  MoveL 7660 to (-403.64, 335.28, -48.3) mm, rotated rx -180 ry 0 rz 0.01 deg; joints [35.458, -30.408, 74.668, -134.792, 54.854, 150.831]
  MoveL 7661 to (-403.75, 334.45, -48.33) mm, rotated rx -180 ry 0 rz 0.01 deg; joints [35.434, -30.43, 74.717, -134.831, 54.861, 150.87]
  MoveL 7662 to (-403.78, 333.95, -48.34) mm, rotated rx -180 ry 0 rz 0.01 deg; joints [35.42, -30.445, 74.752, -134.855, 54.867, 150.895]
  MoveL 7663 to (-403.79, 333.65, -48.35) mm, rotated rx -180 ry 0 rz 0.01 deg; joints [35.412, -30.454, 74.772, -134.869, 54.871, 150.909]
  MoveL 7664 to (-403.79, 333.1, -48.37) mm, rotated rx -180 ry 0 rz 0.01 deg; joints [35.398, -30.473, 74.813, -134.896, 54.879, 150.938]
  MoveL 7665 to (-401.27, 328.17, -48.57) mm, rotated rx -180 ry 0 rz 0.01 deg; joints [35.314, -30.758, 75.431, -135.148, 55.073, 151.276]
  MoveL 7666 to (-395.8, 327.3, -48.77) mm, rotated rx 180 ry 0 rz 0.01 deg; joints [35.394, -31.047, 76.052, -135.227, 55.349, 151.512]
  MoveL 7667 to (-391.89, 331.22, -48.97) mm, rotated rx 180 ry 0 rz 0.01 deg; joints [35.572, -31.096, 76.166, -135.071, 55.483, 151.459]
  MoveL 7668 to (-392.75, 336.69, -49.18) mm, rotated rx -180 ry 0 rz 0.01 deg; joints [35.7, -30.858, 75.678, -134.814, 55.371, 151.167]
  MoveL 7669 to (-397.69, 339.2, -49.38) mm, rotated rx 180 ry 0 rz 0.01 deg; joints [35.673, -30.52, 74.987, -134.669, 55.109, 150.878]
  MoveL 7670 to (-398.51, 339.2, -49.4) mm, rotated rx -180 ry 0 rz 0.01 deg; joints [35.658, -30.478, 74.902, -134.664, 55.071, 150.85]
  MoveL 7671 to (-399.34, 339.13, -49.43) mm, rotated rx 180 ry 0 rz 0.01 deg; joints [35.641, -30.438, 74.822, -134.661, 55.033, 150.826]
  MoveL 7672 to (-399.55, 339.1, -49.44) mm, rotated rx -180 ry 0 rz 0.01 deg; joints [35.636, -30.428, 74.802, -134.662, 55.024, 150.82]
  MoveL 7673 to (-402.87, 337.02, -49.58) mm, rotated rx -180 ry 0 rz 0.01 deg; joints [35.519, -30.33, 74.612, -134.739, 54.9, 150.812]
  MoveL 7674 to (-402.89, 336.99, -49.58) mm, rotated rx -180 ry 0 rz 0.01 deg; joints [35.517, -30.33, 74.612, -134.74, 54.899, 150.813]
  MoveL 7675 to (-403.36, 336.14, -49.62) mm, rotated rx 180 ry 0 rz 0.01 deg; joints [35.486, -30.334, 74.625, -134.777, 54.89, 150.84]
  MoveL 7676 to (-403.42, 336, -49.62) mm, rotated rx -180 ry 0 rz 0.01 deg; joints [35.482, -30.336, 74.629, -134.784, 54.889, 150.845]
  MoveL 7677 to (-403.6, 335.45, -49.64) mm, rotated rx -180 ry 0 rz 0.01 deg; joints [35.464, -30.345, 74.651, -134.809, 54.889, 150.867]
  MoveL 7678 to (-403.64, 335.28, -49.65) mm, rotated rx -180 ry 0 rz 0.01 deg; joints [35.459, -30.349, 74.659, -134.817, 54.889, 150.874]
  MoveL 7679 to (-403.75, 334.45, -49.68) mm, rotated rx -180 ry 0 rz 0.01 deg; joints [35.434, -30.371, 74.709, -134.856, 54.896, 150.913]
  MoveL 7680 to (-403.78, 333.95, -49.7) mm, rotated rx -180 ry 0 rz 0.01 deg; joints [35.421, -30.386, 74.743, -134.88, 54.903, 150.938]
  MoveL 7681 to (-403.79, 333.65, -49.71) mm, rotated rx 180 ry 0 rz 0.01 deg; joints [35.413, -30.396, 74.764, -134.894, 54.907, 150.952]
  MoveL 7682 to (-403.79, 333.1, -49.72) mm, rotated rx -180 ry 0 rz 0.01 deg; joints [35.398, -30.414, 74.804, -134.92, 54.915, 150.981]
  MoveL 7683 to (-401.27, 328.17, -49.93) mm, rotated rx 180 ry 0 rz 0.01 deg; joints [35.315, -30.699, 75.423, -135.172, 55.109, 151.319]
  MoveL 7684 to (-395.8, 327.3, -50.13) mm, rotated rx 180 ry 0 rz 0.01 deg; joints [35.395, -30.988, 76.044, -135.25, 55.385, 151.555]
  MoveL 7685 to (-391.89, 331.22, -50.33) mm, rotated rx 180 ry 0 rz 0.01 deg; joints [35.573, -31.037, 76.157, -135.095, 55.519, 151.502]
  MoveL 7686 to (-392.75, 336.69, -50.53) mm, rotated rx -180 ry 0 rz 0.01 deg; joints [35.701, -30.799, 75.67, -134.838, 55.407, 151.21]
  MoveL 7687 to (-397.69, 339.2, -50.73) mm, rotated rx 180 ry 0 rz 0.01 deg; joints [35.674, -30.461, 74.978, -134.693, 55.144, 150.921]
  MoveL 7688 to (-398.51, 339.2, -50.76) mm, rotated rx 180 ry 0 rz 0.01 deg; joints [35.659, -30.419, 74.894, -134.688, 55.106, 150.894]
  MoveL 7689 to (-399.34, 339.13, -50.79) mm, rotated rx -180 ry 0 rz 0.01 deg; joints [35.641, -30.379, 74.813, -134.686, 55.069, 150.869]
  MoveL 7690 to (-399.55, 339.1, -50.79) mm, rotated rx -180 ry 0 rz 0.01 deg; joints [35.636, -30.369, 74.793, -134.686, 55.059, 150.863]
  MoveL 7691 to (-402.87, 337.02, -50.93) mm, rotated rx -180 ry 0 rz 0.01 deg; joints [35.519, -30.271, 74.603, -134.763, 54.935, 150.855]
  MoveL 7692 to (-402.89, 336.99, -50.94) mm, rotated rx -180 ry 0 rz 0.01 deg; joints [35.518, -30.271, 74.603, -134.765, 54.935, 150.856]
  MoveL 7693 to (-403.36, 336.14, -50.97) mm, rotated rx 180 ry 0 rz 0.01 deg; joints [35.487, -30.276, 74.616, -134.802, 54.925, 150.883]
  MoveL 7694 to (-403.42, 336, -50.97) mm, rotated rx 180 ry 0 rz 0.01 deg; joints [35.482, -30.277, 74.62, -134.808, 54.924, 150.888]
  MoveL 7695 to (-403.6, 335.45, -50.99) mm, rotated rx -180 ry 0 rz 0.01 deg; joints [35.464, -30.287, 74.642, -134.833, 54.924, 150.91]
  MoveL 7696 to (-403.64, 335.28, -51) mm, rotated rx -180 ry 0 rz 0.01 deg; joints [35.459, -30.29, 74.651, -134.841, 54.925, 150.917]
  MoveL 7697 to (-403.75, 334.45, -51.03) mm, rotated rx -180 ry 0 rz 0.01 deg; joints [35.435, -30.312, 74.7, -134.88, 54.932, 150.956]
  MoveL 7698 to (-403.78, 333.95, -51.05) mm, rotated rx -180 ry 0 rz 0.01 deg; joints [35.421, -30.328, 74.734, -134.904, 54.938, 150.98]
  MoveL 7699 to (-403.79, 333.65, -51.06) mm, rotated rx 180 ry 0 rz 0.01 deg; joints [35.413, -30.337, 74.755, -134.918, 54.942, 150.995]
  MoveL 7700 to (-403.79, 333.1, -51.08) mm, rotated rx -180 ry 0 rz 0.01 deg; joints [35.399, -30.355, 74.795, -134.944, 54.951, 151.023]
  MoveL 7701 to (-401.27, 328.17, -51.28) mm, rotated rx 180 ry 0 rz 0.01 deg; joints [35.316, -30.64, 75.414, -135.197, 55.145, 151.362]
  MoveL 7702 to (-395.8, 327.3, -51.48) mm, rotated rx 180 ry 0 rz 0.01 deg; joints [35.396, -30.929, 76.035, -135.274, 55.421, 151.598]
  MoveL 7703 to (-391.89, 331.22, -51.68) mm, rotated rx -180 ry 0 rz 0.01 deg; joints [35.573, -30.978, 76.148, -135.118, 55.555, 151.545]
  MoveL 7704 to (-392.75, 336.69, -51.88) mm, rotated rx 180 ry 0 rz 0.01 deg; joints [35.702, -30.74, 75.661, -134.862, 55.443, 151.253]
  MoveL 7705 to (-397.69, 339.2, -52.08) mm, rotated rx -180 ry 0 rz 0.01 deg; joints [35.675, -30.402, 74.969, -134.717, 55.18, 150.964]
  MoveL 7706 to (-398.51, 339.2, -52.11) mm, rotated rx -180 ry 0 rz 0.01 deg; joints [35.659, -30.36, 74.885, -134.712, 55.142, 150.936]
  MoveL 7707 to (-399.34, 339.13, -52.14) mm, rotated rx -180 ry 0 rz 0.01 deg; joints [35.642, -30.32, 74.804, -134.71, 55.104, 150.912]
  MoveL 7708 to (-399.55, 339.1, -52.15) mm, rotated rx 180 ry 0 rz 0.01 deg; joints [35.637, -30.311, 74.784, -134.71, 55.095, 150.906]
  MoveL 7709 to (-402.87, 337.02, -52.29) mm, rotated rx 180 ry 0 rz 0.01 deg; joints [35.52, -30.212, 74.594, -134.788, 54.971, 150.898]
  MoveL 7710 to (-402.89, 336.99, -52.29) mm, rotated rx -180 ry 0 rz 0.01 deg; joints [35.519, -30.212, 74.594, -134.789, 54.97, 150.899]
  MoveL 7711 to (-403.36, 336.14, -52.32) mm, rotated rx 180 ry 0 rz 0.01 deg; joints [35.488, -30.217, 74.607, -134.826, 54.961, 150.926]
  MoveL 7712 to (-403.42, 336, -52.33) mm, rotated rx -180 ry 0 rz 0.01 deg; joints [35.483, -30.219, 74.611, -134.832, 54.96, 150.931]
  MoveL 7713 to (-403.6, 335.45, -52.35) mm, rotated rx 180 ry 0 rz 0.01 deg; joints [35.465, -30.228, 74.633, -134.857, 54.96, 150.953]
  MoveL 7714 to (-403.64, 335.28, -52.35) mm, rotated rx -180 ry 0 rz 0.01 deg; joints [35.46, -30.231, 74.642, -134.865, 54.96, 150.96]
  MoveL 7715 to (-403.75, 334.45, -52.38) mm, rotated rx -180 ry 0 rz 0.01 deg; joints [35.436, -30.253, 74.691, -134.904, 54.967, 150.999]
  MoveL 7716 to (-403.78, 333.95, -52.4) mm, rotated rx -180 ry 0 rz 0.01 deg; joints [35.422, -30.269, 74.725, -134.928, 54.974, 151.023]
  MoveL 7717 to (-403.79, 333.65, -52.41) mm, rotated rx -180 ry 0 rz 0.01 deg; joints [35.414, -30.278, 74.746, -134.942, 54.978, 151.038]
  MoveL 7718 to (-403.79, 333.1, -52.43) mm, rotated rx -180 ry 0 rz 0.01 deg; joints [35.399, -30.296, 74.786, -134.968, 54.986, 151.066]
  MoveL 7719 to (-401.27, 328.17, -52.63) mm, rotated rx 180 ry 0 rz 0.01 deg; joints [35.316, -30.581, 75.405, -135.22, 55.181, 151.405]
  MoveL 7720 to (-395.8, 327.3, -52.83) mm, rotated rx 180 ry 0 rz 0.01 deg; joints [35.396, -30.87, 76.026, -135.298, 55.457, 151.64]
  MoveL 7721 to (-391.89, 331.22, -53.03) mm, rotated rx -180 ry 0 rz 0.01 deg; joints [35.574, -30.918, 76.139, -135.142, 55.591, 151.588]
  MoveL 7722 to (-392.75, 336.69, -53.23) mm, rotated rx -180 ry 0 rz 0.01 deg; joints [35.702, -30.681, 75.652, -134.886, 55.478, 151.296]
  MoveL 7723 to (-397.69, 339.2, -53.43) mm, rotated rx -180 ry 0 rz 0.01 deg; joints [35.675, -30.343, 74.96, -134.741, 55.215, 151.007]
  MoveL 7724 to (-398.51, 339.2, -53.46) mm, rotated rx -180 ry 0 rz 0.01 deg; joints [35.66, -30.301, 74.876, -134.736, 55.177, 150.979]
  MoveL 7725 to (-399.34, 339.13, -53.49) mm, rotated rx 180 ry 0 rz 0.01 deg; joints [35.642, -30.261, 74.795, -134.734, 55.14, 150.954]
  MoveL 7726 to (-399.55, 339.1, -53.5) mm, rotated rx -180 ry 0 rz 0.01 deg; joints [35.637, -30.252, 74.775, -134.734, 55.13, 150.949]
  MoveL 7727 to (-402.87, 337.02, -53.64) mm, rotated rx -180 ry 0 rz 0.01 deg; joints [35.52, -30.154, 74.585, -134.812, 55.006, 150.941]
  MoveL 7728 to (-402.89, 336.99, -53.64) mm, rotated rx -180 ry 0 rz 0.01 deg; joints [35.519, -30.154, 74.585, -134.813, 55.005, 150.942]
  MoveL 7729 to (-403.36, 336.14, -53.67) mm, rotated rx -180 ry 0 rz 0.01 deg; joints [35.488, -30.158, 74.598, -134.85, 54.996, 150.968]
  MoveL 7730 to (-403.42, 336, -53.68) mm, rotated rx -180 ry 0 rz 0.01 deg; joints [35.483, -30.16, 74.602, -134.856, 54.995, 150.974]
  MoveL 7731 to (-403.6, 335.45, -53.7) mm, rotated rx 180 ry 0 rz 0.01 deg; joints [35.465, -30.169, 74.624, -134.881, 54.995, 150.995]
  MoveL 7732 to (-403.64, 335.28, -53.71) mm, rotated rx -180 ry 0 rz 0.01 deg; joints [35.46, -30.173, 74.633, -134.889, 54.996, 151.003]
  MoveL 7733 to (-403.75, 334.45, -53.74) mm, rotated rx -180 ry 0 rz 0.01 deg; joints [35.436, -30.194, 74.682, -134.928, 55.003, 151.041]
  MoveL 7734 to (-403.78, 333.95, -53.75) mm, rotated rx -180 ry 0 rz 0.01 deg; joints [35.422, -30.21, 74.716, -134.952, 55.009, 151.066]
  MoveL 7735 to (-403.79, 333.65, -53.76) mm, rotated rx -180 ry 0 rz 0.01 deg; joints [35.415, -30.219, 74.737, -134.966, 55.013, 151.081]
  MoveL 7736 to (-403.79, 333.1, -53.78) mm, rotated rx -180 ry 0 rz 0.01 deg; joints [35.4, -30.237, 74.777, -134.992, 55.022, 151.109]
  MoveL 7737 to (-401.27, 328.17, -53.98) mm, rotated rx -180 ry 0 rz 0.01 deg; joints [35.317, -30.522, 75.396, -135.244, 55.217, 151.447]
  MoveL 7738 to (-395.8, 327.3, -54.18) mm, rotated rx 180 ry 0 rz 0.01 deg; joints [35.397, -30.811, 76.017, -135.322, 55.493, 151.683]
  MoveL 7739 to (-391.89, 331.22, -54.38) mm, rotated rx 180 ry 0 rz 0.01 deg; joints [35.575, -30.859, 76.13, -135.166, 55.627, 151.63]
  MoveL 7740 to (-392.75, 336.69, -54.59) mm, rotated rx -180 ry 0 rz 0.01 deg; joints [35.703, -30.621, 75.643, -134.91, 55.514, 151.339]
  MoveL 7741 to (-397.69, 339.2, -54.79) mm, rotated rx -180 ry 0 rz 0.01 deg; joints [35.676, -30.284, 74.951, -134.765, 55.251, 151.05]
  MoveL 7742 to (-398.51, 339.2, -54.81) mm, rotated rx -180 ry 0 rz 0.01 deg; joints [35.66, -30.242, 74.866, -134.76, 55.213, 151.022]
  MoveL 7743 to (-399.34, 339.13, -54.84) mm, rotated rx -180 ry 0 rz 0.01 deg; joints [35.643, -30.202, 74.786, -134.758, 55.175, 150.997]
  MoveL 7744 to (-399.55, 339.1, -54.85) mm, rotated rx -180 ry 0 rz 0.01 deg; joints [35.638, -30.193, 74.766, -134.758, 55.165, 150.992]
  MoveL 7745 to (-402.87, 337.02, -54.99) mm, rotated rx 180 ry 0 rz 0.01 deg; joints [35.521, -30.095, 74.576, -134.836, 55.041, 150.984]
  MoveL 7746 to (-402.89, 336.99, -54.99) mm, rotated rx -180 ry 0 rz 0.01 deg; joints [35.52, -30.095, 74.576, -134.837, 55.041, 150.984]
  MoveL 7747 to (-403.36, 336.14, -55.03) mm, rotated rx -180 ry 0 rz 0.01 deg; joints [35.489, -30.099, 74.589, -134.874, 55.031, 151.011]
  MoveL 7748 to (-403.42, 336, -55.03) mm, rotated rx 180 ry 0 rz 0.01 deg; joints [35.484, -30.101, 74.593, -134.88, 55.031, 151.016]
  MoveL 7749 to (-403.6, 335.45, -55.05) mm, rotated rx 180 ry 0 rz 0.01 deg; joints [35.466, -30.11, 74.615, -134.905, 55.03, 151.038]
  MoveL 7750 to (-403.64, 335.28, -55.06) mm, rotated rx 180 ry 0 rz 0.01 deg; joints [35.461, -30.114, 74.623, -134.913, 55.031, 151.045]
  MoveL 7751 to (-403.75, 334.45, -55.09) mm, rotated rx -180 ry 0 rz 0.01 deg; joints [35.437, -30.135, 74.673, -134.952, 55.038, 151.084]
  MoveL 7752 to (-403.78, 333.95, -55.11) mm, rotated rx -180 ry 0 rz 0.01 deg; joints [35.423, -30.151, 74.707, -134.976, 55.045, 151.109]
  MoveL 7753 to (-403.79, 333.65, -55.12) mm, rotated rx -180 ry 0 rz 0.01 deg; joints [35.415, -30.16, 74.727, -134.99, 55.049, 151.123]
  MoveL 7754 to (-403.79, 333.1, -55.14) mm, rotated rx -180 ry 0 rz 0.01 deg; joints [35.401, -30.178, 74.768, -135.016, 55.057, 151.151]
  MoveL 7755 to (-401.27, 328.17, -55.34) mm, rotated rx -180 ry 0 rz 0.01 deg; joints [35.317, -30.463, 75.387, -135.268, 55.252, 151.49]
  MoveL 7756 to (-395.8, 327.3, -55.54) mm, rotated rx -180 ry 0 rz 0.01 deg; joints [35.397, -30.751, 76.008, -135.345, 55.529, 151.725]
  MoveL 7757 to (-391.89, 331.22, -55.74) mm, rotated rx -180 ry 0 rz 0.01 deg; joints [35.575, -30.8, 76.121, -135.189, 55.663, 151.673]
  MoveL 7758 to (-392.75, 336.69, -55.94) mm, rotated rx 180 ry 0 rz 0.01 deg; joints [35.703, -30.562, 75.633, -134.934, 55.55, 151.381]
  MoveL 7759 to (-397.69, 339.2, -56.14) mm, rotated rx -180 ry 0 rz 0.01 deg; joints [35.676, -30.225, 74.942, -134.789, 55.286, 151.092]
  MoveL 7760 to (-398.51, 339.2, -56.17) mm, rotated rx -180 ry 0 rz 0.01 deg; joints [35.661, -30.183, 74.857, -134.784, 55.248, 151.065]
  MoveL 7761 to (-399.34, 339.13, -56.2) mm, rotated rx 180 ry 0 rz 0.01 deg; joints [35.644, -30.143, 74.776, -134.782, 55.21, 151.04]
  MoveL 7762 to (-399.55, 339.1, -56.2) mm, rotated rx 180 ry 0 rz 0.01 deg; joints [35.639, -30.134, 74.756, -134.782, 55.201, 151.034]
  MoveL 7763 to (-402.87, 337.02, -56.34) mm, rotated rx -180 ry 0 rz 0.01 deg; joints [35.522, -30.036, 74.566, -134.86, 55.076, 151.026]
  MoveL 7764 to (-402.89, 336.99, -56.35) mm, rotated rx -180 ry 0 rz 0.01 deg; joints [35.52, -30.036, 74.566, -134.861, 55.076, 151.027]
  MoveL 7765 to (-403.36, 336.14, -56.38) mm, rotated rx -180 ry 0 rz 0.01 deg; joints [35.489, -30.04, 74.58, -134.898, 55.067, 151.054]
  MoveL 7766 to (-403.42, 336, -56.38) mm, rotated rx 180 ry 0 rz 0.01 deg; joints [35.484, -30.042, 74.584, -134.904, 55.066, 151.059]
  MoveL 7767 to (-403.6, 335.45, -56.4) mm, rotated rx -180 ry 0 rz 0.01 deg; joints [35.467, -30.051, 74.605, -134.929, 55.066, 151.08]
  MoveL 7768 to (-403.64, 335.28, -56.41) mm, rotated rx -180 ry 0 rz 0.01 deg; joints [35.461, -30.055, 74.614, -134.937, 55.066, 151.088]
  MoveL 7769 to (-403.75, 334.45, -56.44) mm, rotated rx -180 ry 0 rz 0.01 deg; joints [35.437, -30.076, 74.663, -134.976, 55.074, 151.126]
  MoveL 7770 to (-403.78, 333.95, -56.46) mm, rotated rx -180 ry 0 rz 0.01 deg; joints [35.424, -30.092, 74.697, -135, 55.08, 151.151]
  MoveL 7771 to (-403.79, 333.65, -56.47) mm, rotated rx -180 ry 0 rz 0.01 deg; joints [35.416, -30.101, 74.718, -135.014, 55.084, 151.166]
  MoveL 7772 to (-403.79, 333.1, -56.49) mm, rotated rx 180 ry 0 rz 0.01 deg; joints [35.401, -30.119, 74.758, -135.04, 55.093, 151.194]
  MoveL 7773 to (-401.27, 328.17, -56.69) mm, rotated rx 180 ry 0 rz 0.01 deg; joints [35.318, -30.404, 75.377, -135.292, 55.288, 151.532]
  MoveL 7774 to (-395.8, 327.3, -56.89) mm, rotated rx -180 ry 0 rz 0.01 deg; joints [35.398, -30.692, 75.998, -135.369, 55.565, 151.768]
  MoveL 7775 to (-391.89, 331.22, -57.09) mm, rotated rx 180 ry 0 rz 0.01 deg; joints [35.576, -30.74, 76.112, -135.213, 55.699, 151.715]
  MoveL 7776 to (-392.75, 336.69, -57.29) mm, rotated rx 180 ry 0 rz 0.01 deg; joints [35.704, -30.503, 75.624, -134.957, 55.585, 151.424]
  MoveL 7777 to (-397.69, 339.2, -57.49) mm, rotated rx -180 ry 0 rz 0.01 deg; joints [35.677, -30.166, 74.932, -134.813, 55.321, 151.135]
  MoveL 7778 to (-398.51, 339.2, -57.52) mm, rotated rx -180 ry 0 rz 0.01 deg; joints [35.661, -30.124, 74.847, -134.808, 55.283, 151.107]
  MoveL 7779 to (-399.34, 339.13, -57.55) mm, rotated rx 180 ry 0 rz 0.01 deg; joints [35.644, -30.084, 74.767, -134.806, 55.245, 151.082]
  MoveL 7780 to (-399.55, 339.1, -57.56) mm, rotated rx -180 ry 0 rz 0.01 deg; joints [35.639, -30.074, 74.747, -134.806, 55.236, 151.077]
  MoveL 7781 to (-402.87, 337.02, -57.7) mm, rotated rx -180 ry 0 rz 0.01 deg; joints [35.522, -29.976, 74.556, -134.884, 55.112, 151.068]
  MoveL 7782 to (-402.89, 336.99, -57.7) mm, rotated rx -180 ry 0 rz 0.01 deg; joints [35.521, -29.976, 74.556, -134.885, 55.111, 151.069]
  MoveL 7783 to (-403.36, 336.14, -57.73) mm, rotated rx -180 ry 0 rz 0.01 deg; joints [35.49, -29.981, 74.57, -134.922, 55.102, 151.096]
  MoveL 7784 to (-403.42, 336, -57.74) mm, rotated rx -180 ry 0 rz 0.01 deg; joints [35.485, -29.983, 74.574, -134.928, 55.101, 151.101]
  MoveL 7785 to (-403.6, 335.45, -57.76) mm, rotated rx -180 ry 0 rz 0.01 deg; joints [35.467, -29.992, 74.596, -134.953, 55.101, 151.123]
  MoveL 7786 to (-403.64, 335.28, -57.76) mm, rotated rx 180 ry 0 rz 0.01 deg; joints [35.462, -29.995, 74.604, -134.961, 55.102, 151.13]
  MoveL 7787 to (-403.75, 334.45, -57.79) mm, rotated rx -180 ry 0 rz 0.01 deg; joints [35.438, -30.017, 74.654, -135, 55.109, 151.169]
  MoveL 7788 to (-403.78, 333.95, -57.81) mm, rotated rx -180 ry 0 rz 0.01 deg; joints [35.424, -30.033, 74.688, -135.024, 55.115, 151.193]
  MoveL 7789 to (-403.79, 333.65, -57.82) mm, rotated rx -180 ry 0 rz 0.01 deg; joints [35.416, -30.042, 74.708, -135.038, 55.119, 151.208]
  MoveL 7790 to (-403.79, 333.1, -57.84) mm, rotated rx -180 ry 0 rz 0.01 deg; joints [35.402, -30.06, 74.749, -135.064, 55.128, 151.236]
  MoveL 7791 to (-401.27, 328.17, -58.04) mm, rotated rx -180 ry 0 rz 0.01 deg; joints [35.319, -30.344, 75.368, -135.315, 55.324, 151.574]
  MoveL 7792 to (-395.8, 327.3, -58.24) mm, rotated rx 180 ry 0 rz 0.01 deg; joints [35.399, -30.632, 75.989, -135.392, 55.601, 151.81]
  MoveL 7793 to (-391.89, 331.22, -58.44) mm, rotated rx -180 ry 0 rz 0.01 deg; joints [35.576, -30.681, 76.102, -135.236, 55.734, 151.757]
  MoveL 7794 to (-392.75, 336.69, -58.64) mm, rotated rx 180 ry 0 rz 0.01 deg; joints [35.705, -30.443, 75.614, -134.981, 55.621, 151.466]
  MoveL 7795 to (-397.69, 339.2, -58.84) mm, rotated rx 180 ry 0 rz 0.01 deg; joints [35.677, -30.106, 74.922, -134.836, 55.356, 151.177]
  MoveL 7796 to (-398.51, 339.2, -58.87) mm, rotated rx -180 ry 0 rz 0.01 deg; joints [35.662, -30.065, 74.838, -134.831, 55.318, 151.149]
  MoveL 7797 to (-399.34, 339.13, -58.9) mm, rotated rx -180 ry 0 rz 0.01 deg; joints [35.645, -30.025, 74.757, -134.829, 55.281, 151.125]
  MoveL 7798 to (-399.55, 339.1, -58.91) mm, rotated rx -180 ry 0 rz 0.01 deg; joints [35.64, -30.015, 74.737, -134.83, 55.271, 151.119]
  MoveL 7799 to (-402.87, 337.02, -59.05) mm, rotated rx 180 ry 0 rz 0.01 deg; joints [35.523, -29.917, 74.547, -134.907, 55.147, 151.111]
  MoveL 7800 to (-402.89, 336.99, -59.05) mm, rotated rx -180 ry 0 rz 0.01 deg; joints [35.522, -29.917, 74.547, -134.909, 55.146, 151.112]
  MoveL 7801 to (-403.36, 336.14, -59.08) mm, rotated rx -180 ry 0 rz 0.01 deg; joints [35.491, -29.922, 74.56, -134.946, 55.137, 151.138]
  MoveL 7802 to (-403.42, 336, -59.09) mm, rotated rx -180 ry 0 rz 0.01 deg; joints [35.486, -29.923, 74.564, -134.952, 55.136, 151.143]
  MoveL 7803 to (-403.6, 335.45, -59.11) mm, rotated rx -180 ry 0 rz 0.01 deg; joints [35.468, -29.933, 74.586, -134.977, 55.136, 151.165]
  MoveL 7804 to (-403.64, 335.28, -59.12) mm, rotated rx -180 ry 0 rz 0.01 deg; joints [35.463, -29.936, 74.594, -134.985, 55.137, 151.172]
  MoveL 7805 to (-403.75, 334.45, -59.15) mm, rotated rx -180 ry 0 rz 0.01 deg; joints [35.438, -29.958, 74.644, -135.024, 55.144, 151.211]
  MoveL 7806 to (-403.78, 333.95, -59.16) mm, rotated rx -180 ry 0 rz 0.01 deg; joints [35.425, -29.973, 74.678, -135.047, 55.151, 151.236]
  MoveL 7807 to (-403.79, 333.65, -59.17) mm, rotated rx -180 ry 0 rz 0.01 deg; joints [35.417, -29.983, 74.699, -135.061, 55.155, 151.25]
  MoveL 7808 to (-403.79, 333.1, -59.19) mm, rotated rx -180 ry 0 rz 0.01 deg; joints [35.402, -30.001, 74.739, -135.088, 55.163, 151.278]
  MoveL 7809 to (-401.27, 328.17, -59.39) mm, rotated rx 180 ry 0 rz 0.01 deg; joints [35.319, -30.285, 75.358, -135.339, 55.359, 151.616]
  MoveL 7810 to (-395.8, 327.3, -59.59) mm, rotated rx 180 ry 0 rz 0.01 deg; joints [35.399, -30.573, 75.979, -135.416, 55.636, 151.852]
  MoveL 7811 to (-391.89, 331.22, -59.79) mm, rotated rx 180 ry 0 rz 0.01 deg; joints [35.577, -30.621, 76.092, -135.259, 55.77, 151.8]
  MoveL 7812 to (-392.75, 336.69, -60) mm, rotated rx -180 ry 0 rz 0.01 deg; joints [35.705, -30.384, 75.604, -135.004, 55.656, 151.508]
  MoveL 7813 to (-397.69, 339.2, -60.2) mm, rotated rx -180 ry 0 rz 0.01 deg; joints [35.678, -30.047, 74.912, -134.86, 55.391, 151.219]
  MoveL 7814 to (-398.51, 339.2, -60.22) mm, rotated rx -180 ry 0 rz 0.01 deg; joints [35.663, -30.006, 74.828, -134.855, 55.353, 151.192]
  MoveL 7815 to (-399.34, 339.13, -60.25) mm, rotated rx 180 ry 0 rz 0.01 deg; joints [35.645, -29.966, 74.747, -134.853, 55.316, 151.167]
  MoveL 7816 to (-399.55, 339.1, -60.26) mm, rotated rx -180 ry 0 rz 0.01 deg; joints [35.64, -29.956, 74.727, -134.853, 55.306, 151.161]
  MoveL 7817 to (-402.87, 337.02, -60.4) mm, rotated rx 180 ry 0 rz 0.01 deg; joints [35.523, -29.858, 74.537, -134.931, 55.182, 151.153]
  MoveL 7818 to (-402.89, 336.99, -60.4) mm, rotated rx -180 ry 0 rz 0.01 deg; joints [35.522, -29.858, 74.537, -134.932, 55.181, 151.154]
  MoveL 7819 to (-403.36, 336.14, -60.44) mm, rotated rx -180 ry 0 rz 0.01 deg; joints [35.491, -29.862, 74.55, -134.969, 55.172, 151.18]
  MoveL 7820 to (-403.42, 336, -60.44) mm, rotated rx -180 ry 0 rz 0.01 deg; joints [35.486, -29.864, 74.554, -134.976, 55.171, 151.186]
  MoveL 7821 to (-403.6, 335.45, -60.46) mm, rotated rx -180 ry 0 rz 0.01 deg; joints [35.468, -29.873, 74.576, -135.001, 55.171, 151.207]
  MoveL 7822 to (-403.64, 335.28, -60.47) mm, rotated rx -180 ry 0 rz 0.01 deg; joints [35.463, -29.877, 74.584, -135.008, 55.172, 151.214]
  MoveL 7823 to (-403.75, 334.45, -60.5) mm, rotated rx -180 ry 0 rz 0.01 deg; joints [35.439, -29.899, 74.634, -135.047, 55.179, 151.253]
  MoveL 7824 to (-403.78, 333.95, -60.52) mm, rotated rx -180 ry 0 rz 0.01 deg; joints [35.425, -29.914, 74.668, -135.071, 55.186, 151.278]
  MoveL 7825 to (-403.79, 333.65, -60.53) mm, rotated rx -180 ry 0 rz 0.01 deg; joints [35.417, -29.923, 74.689, -135.085, 55.19, 151.292]
  MoveL 7826 to (-403.79, 333.1, -60.55) mm, rotated rx -180 ry 0 rz 0.01 deg; joints [35.403, -29.941, 74.729, -135.111, 55.199, 151.32]
  MoveL 7827 to (-401.27, 328.17, -60.75) mm, rotated rx -180 ry 0 rz 0.01 deg; joints [35.32, -30.225, 75.348, -135.362, 55.395, 151.658]
  MoveL 7828 to (-395.8, 327.3, -60.95) mm, rotated rx 180 ry 0 rz 0.01 deg; joints [35.4, -30.513, 75.969, -135.439, 55.672, 151.894]
  MoveL 7829 to (-391.89, 331.22, -61.15) mm, rotated rx 180 ry 0 rz 0.01 deg; joints [35.578, -30.561, 76.082, -135.283, 55.806, 151.842]
  MoveL 7830 to (-392.75, 336.69, -61.35) mm, rotated rx 180 ry 0 rz 0.01 deg; joints [35.706, -30.324, 75.594, -135.027, 55.691, 151.55]
  MoveL 7831 to (-397.69, 339.2, -61.55) mm, rotated rx 180 ry 0 rz 0.01 deg; joints [35.679, -29.988, 74.902, -134.883, 55.427, 151.262]
  MoveL 7832 to (-398.51, 339.2, -61.58) mm, rotated rx -180 ry 0 rz 0.01 deg; joints [35.663, -29.946, 74.818, -134.878, 55.388, 151.234]
  MoveL 7833 to (-399.34, 339.13, -61.61) mm, rotated rx 180 ry 0 rz 0.01 deg; joints [35.646, -29.906, 74.737, -134.877, 55.351, 151.209]
  MoveL 7834 to (-399.55, 339.1, -61.61) mm, rotated rx -180 ry 0 rz 0.01 deg; joints [35.641, -29.896, 74.717, -134.877, 55.341, 151.203]
  MoveL 7835 to (-402.87, 337.02, -61.75) mm, rotated rx -180 ry 0 rz 0.01 deg; joints [35.524, -29.799, 74.527, -134.955, 55.217, 151.195]
  MoveL 7836 to (-402.89, 336.99, -61.76) mm, rotated rx 180 ry 0 rz 0.01 deg; joints [35.523, -29.799, 74.527, -134.956, 55.217, 151.196]
  MoveL 7837 to (-403.36, 336.14, -61.79) mm, rotated rx -180 ry 0 rz 0.01 deg; joints [35.492, -29.803, 74.54, -134.993, 55.207, 151.222]
  MoveL 7838 to (-403.42, 336, -61.79) mm, rotated rx 180 ry 0 rz 0.01 deg; joints [35.487, -29.805, 74.544, -134.999, 55.207, 151.228]
  MoveL 7839 to (-403.6, 335.45, -61.82) mm, rotated rx -180 ry 0 rz 0.01 deg; joints [35.469, -29.814, 74.566, -135.024, 55.206, 151.249]
  MoveL 7840 to (-403.64, 335.28, -61.82) mm, rotated rx -180 ry 0 rz 0.01 deg; joints [35.464, -29.818, 74.574, -135.032, 55.207, 151.257]
  MoveL 7841 to (-403.75, 334.45, -61.85) mm, rotated rx -180 ry 0 rz 0.01 deg; joints [35.44, -29.839, 74.624, -135.071, 55.215, 151.295]
  MoveL 7842 to (-403.78, 333.95, -61.87) mm, rotated rx -180 ry 0 rz 0.01 deg; joints [35.426, -29.855, 74.658, -135.095, 55.221, 151.32]
  MoveL 7843 to (-403.79, 333.65, -61.88) mm, rotated rx -180 ry 0 rz 0.01 deg; joints [35.418, -29.864, 74.678, -135.109, 55.225, 151.334]
  MoveL 7844 to (-403.79, 333.1, -61.9) mm, rotated rx -180 ry 0 rz 0.01 deg; joints [35.403, -29.882, 74.719, -135.135, 55.234, 151.362]
  MoveL 7845 to (-401.27, 328.17, -62.1) mm, rotated rx 180 ry 0 rz 0.01 deg; joints [35.32, -30.166, 75.338, -135.386, 55.43, 151.7]
  MoveL 7846 to (-395.8, 327.3, -62.3) mm, rotated rx -180 ry 0 rz 0.01 deg; joints [35.4, -30.453, 75.959, -135.462, 55.708, 151.936]
  MoveL 7847 to (-391.89, 331.22, -62.5) mm, rotated rx 180 ry 0 rz 0.01 deg; joints [35.578, -30.502, 76.072, -135.306, 55.841, 151.883]
  MoveL 7848 to (-392.75, 336.69, -62.7) mm, rotated rx -180 ry 0 rz 0.01 deg; joints [35.706, -30.264, 75.584, -135.051, 55.727, 151.592]
  MoveL 7849 to (-397.69, 339.2, -62.9) mm, rotated rx 180 ry 0 rz 0.01 deg; joints [35.679, -29.928, 74.892, -134.907, 55.462, 151.304]
  MoveL 7850 to (-398.51, 339.2, -62.93) mm, rotated rx -180 ry 0 rz 0.01 deg; joints [35.664, -29.887, 74.808, -134.902, 55.424, 151.276]
  MoveL 7851 to (-399.34, 339.13, -62.96) mm, rotated rx -180 ry 0 rz 0.01 deg; joints [35.646, -29.847, 74.727, -134.9, 55.386, 151.251]
  MoveL 7852 to (-399.55, 339.1, -62.97) mm, rotated rx -180 ry 0 rz 0.01 deg; joints [35.641, -29.837, 74.707, -134.9, 55.376, 151.245]
  MoveL 7853 to (-402.87, 337.02, -63.11) mm, rotated rx -180 ry 0 rz 0.01 deg; joints [35.524, -29.739, 74.516, -134.978, 55.252, 151.237]
  MoveL 7854 to (-402.89, 336.99, -63.11) mm, rotated rx -180 ry 0 rz 0.01 deg; joints [35.523, -29.739, 74.516, -134.979, 55.252, 151.238]
  MoveL 7855 to (-403.36, 336.14, -63.14) mm, rotated rx -180 ry 0 rz 0.01 deg; joints [35.492, -29.744, 74.53, -135.016, 55.242, 151.264]
  MoveL 7856 to (-403.42, 336, -63.15) mm, rotated rx -180 ry 0 rz 0.01 deg; joints [35.487, -29.745, 74.534, -135.023, 55.242, 151.27]
  MoveL 7857 to (-403.6, 335.45, -63.17) mm, rotated rx -180 ry 0 rz 0.01 deg; joints [35.47, -29.755, 74.556, -135.048, 55.242, 151.291]
  MoveL 7858 to (-403.64, 335.28, -63.17) mm, rotated rx 180 ry 0 rz 0.01 deg; joints [35.464, -29.758, 74.564, -135.055, 55.242, 151.298]
  MoveL 7859 to (-403.75, 334.45, -63.2) mm, rotated rx -180 ry 0 rz 0.01 deg; joints [35.44, -29.78, 74.613, -135.094, 55.25, 151.337]
  MoveL 7860 to (-403.78, 333.95, -63.22) mm, rotated rx 180 ry 0 rz 0.01 deg; joints [35.426, -29.795, 74.647, -135.118, 55.256, 151.362]
  MoveL 7861 to (-403.79, 333.65, -63.23) mm, rotated rx -180 ry 0 rz 0.01 deg; joints [35.419, -29.804, 74.668, -135.132, 55.26, 151.376]
  MoveL 7862 to (-403.79, 333.1, -63.25) mm, rotated rx 180 ry 0 rz 0.01 deg; joints [35.404, -29.823, 74.709, -135.158, 55.269, 151.404]
  MoveL 7863 to (-401.27, 328.17, -63.45) mm, rotated rx -180 ry 0 rz 0.01 deg; joints [35.321, -30.106, 75.328, -135.409, 55.466, 151.742]
  MoveL 7864 to (-395.8, 327.3, -63.65) mm, rotated rx -180 ry 0 rz 0.01 deg; joints [35.401, -30.393, 75.949, -135.485, 55.743, 151.977]
  MoveL 7865 to (-391.89, 331.22, -63.85) mm, rotated rx -180 ry 0 rz 0.01 deg; joints [35.579, -30.442, 76.062, -135.329, 55.877, 151.925]
  MoveL 7866 to (-392.75, 336.69, -64.05) mm, rotated rx -180 ry 0 rz 0.01 deg; joints [35.707, -30.205, 75.574, -135.074, 55.762, 151.634]
  MoveL 7867 to (-397.69, 339.2, -64.25) mm, rotated rx -180 ry 0 rz 0.01 deg; joints [35.68, -29.869, 74.882, -134.93, 55.497, 151.345]
  MoveL 7868 to (-398.51, 339.2, -64.28) mm, rotated rx -180 ry 0 rz 0.01 deg; joints [35.664, -29.827, 74.797, -134.925, 55.459, 151.318]
  MoveL 7869 to (-399.34, 339.13, -64.31) mm, rotated rx -180 ry 0 rz 0.01 deg; joints [35.647, -29.787, 74.716, -134.923, 55.421, 151.293]
  MoveL 7870 to (-399.55, 339.1, -64.32) mm, rotated rx -180 ry 0 rz 0.01 deg; joints [35.642, -29.778, 74.696, -134.924, 55.411, 151.287]
  MoveL 7871 to (-402.87, 337.02, -64.46) mm, rotated rx -180 ry 0 rz 0.01 deg; joints [35.525, -29.68, 74.506, -135.002, 55.287, 151.279]
  MoveL 7872 to (-402.89, 336.99, -64.46) mm, rotated rx -180 ry 0 rz 0.01 deg; joints [35.524, -29.68, 74.506, -135.003, 55.286, 151.28]
  MoveL 7873 to (-403.36, 336.14, -64.49) mm, rotated rx -180 ry 0 rz 0.01 deg; joints [35.493, -29.684, 74.519, -135.04, 55.277, 151.306]
  MoveL 7874 to (-403.42, 336, -64.5) mm, rotated rx -180 ry 0 rz 0.01 deg; joints [35.488, -29.686, 74.523, -135.046, 55.277, 151.311]
  MoveL 7875 to (-403.53, 335.74, -64.5) mm, rotated rx -180 ry 0 rz 0.01 deg; joints [35.479, -29.689, 74.531, -135.058, 55.275, 151.321]
  MoveL 7876 to (-403.73, 334.87, -64.5) mm, rotated rx 180 ry 0 rz 0.01 deg; joints [35.452, -29.709, 74.575, -135.097, 55.278, 151.357]
  MoveL 7877 to (-403.79, 333.8, -64.5) mm, rotated rx -180 ry 0 rz 0.01 deg; joints [35.423, -29.744, 74.648, -135.147, 55.291, 151.408]
  MoveL 7878 to (-403.78, 32.07, -64.5) mm, rotated rx -180 ry 0 rz 0.01 deg; joints [26.668, -37.864, 92.37, -148.533, 59.34, 163.736]
  MoveL 7879 to (-402.84, 36.1, -64.5) mm, rotated rx -180 ry 0 rz 0.01 deg; joints [26.811, -37.821, 92.27, -148.358, 59.334, 163.62]
  MoveL 7880 to (-402.68, 36.59, -64.5) mm, rotated rx -180 ry 0 rz 0.01 deg; joints [26.829, -37.817, 92.261, -148.336, 59.336, 163.606]
  MoveL 7881 to (-401.99, 38.31, -64.5) mm, rotated rx -180 ry 0 rz 0.01 deg; joints [26.894, -37.811, 92.245, -148.26, 59.347, 163.562]
  MoveL 7882 to (-401.78, 38.75, -64.5) mm, rotated rx -180 ry 0 rz 0.01 deg; joints [26.911, -37.811, 92.244, -148.241, 59.352, 163.552]
  MoveL 7883 to (-396.45, 47.93, -64.5) mm, rotated rx 180 ry 0 rz 0.01 deg; joints [27.287, -37.846, 92.303, -147.834, 59.488, 163.351]
  MoveL 7884 to (-396.1, 48.42, -64.5) mm, rotated rx -180 ry 0 rz 0.01 deg; joints [27.308, -37.851, 92.312, -147.812, 59.498, 163.342]
  MoveL 7885 to (-393.34, 51.68, -64.5) mm, rotated rx 180 ry 0 rz 0.01 deg; joints [27.456, -37.899, 92.411, -147.664, 59.586, 163.289]
  MoveL 7886 to (-393.24, 51.79, -64.5) mm, rotated rx -180 ry 0 rz 0.01 deg; joints [27.461, -37.901, 92.415, -147.659, 59.589, 163.287]
  MoveL 7887 to (-392.24, 52.87, -64.5) mm, rotated rx 180 ry 0 rz 0.01 deg; joints [27.512, -37.921, 92.455, -147.61, 59.622, 163.271]
  MoveL 7888 to (-392.06, 53.05, -64.5) mm, rotated rx 180 ry 0 rz 0.01 deg; joints [27.52, -37.925, 92.463, -147.602, 59.629, 163.269]
  MoveL 7889 to (-389.15, 55.74, -64.5) mm, rotated rx -180 ry 0 rz 0.01 deg; joints [27.653, -37.991, 92.6, -147.479, 59.73, 163.238]
  MoveL 7890 to (-388.93, 55.93, -64.5) mm, rotated rx -180 ry 0 rz 0.01 deg; joints [27.662, -37.996, 92.612, -147.47, 59.738, 163.237]
  MoveL 7891 to (-386.02, 58.18, -64.5) mm, rotated rx 180 ry 0 rz 0.01 deg; joints [27.781, -38.071, 92.769, -147.365, 59.844, 163.221]
  MoveL 7892 to (-385.93, 58.25, -64.5) mm, rotated rx -180 ry 0 rz 0.01 deg; joints [27.785, -38.073, 92.774, -147.362, 59.848, 163.221]
  MoveL 7893 to (-276.03, 137.23, -64.5) mm, rotated rx 180 ry 0 rz 0.01 deg; joints [32.249, -40.718, 98.359, -143.449, 63.678, 162.792]
  MoveL 7894 to (-275.46, 137.56, -64.5) mm, rotated rx -180 ry 0 rz 0.01 deg; joints [32.271, -40.732, 98.389, -143.431, 63.698, 162.792]
  MoveL 7895 to (-273.62, 138.4, -64.5) mm, rotated rx 180 ry 0 rz 0.01 deg; joints [32.333, -40.783, 98.498, -143.382, 63.764, 162.801]
  MoveL 7896 to (-272.9, 138.63, -64.5) mm, rotated rx -180 ry 0 rz 0.01 deg; joints [32.355, -40.804, 98.544, -143.366, 63.791, 162.807]
  MoveL 7897 to (-271.45, 138.94, -64.5) mm, rotated rx 180 ry 0 rz 0.01 deg; joints [32.393, -40.852, 98.648, -143.343, 63.848, 162.826]
  MoveL 7898 to (-270.89, 139, -64.5) mm, rotated rx 180 ry 0 rz 0.01 deg; joints [32.406, -40.872, 98.69, -143.335, 63.87, 162.835]
  MoveL 7899 to (-269.44, 139.06, -64.5) mm, rotated rx 180 ry 0 rz 0.01 deg; joints [32.436, -40.925, 98.807, -143.322, 63.93, 162.862]
  MoveL 7900 to (-268.9, 139.04, -64.5) mm, rotated rx 180 ry 0 rz 0.01 deg; joints [32.446, -40.946, 98.852, -143.318, 63.953, 162.874]
  MoveL 7901 to (-266.73, 138.77, -64.5) mm, rotated rx -180 ry 0 rz 0.01 deg; joints [32.481, -41.034, 99.044, -143.312, 64.048, 162.927]
  MoveL 7902 to (-266.28, 138.69, -64.5) mm, rotated rx -180 ry 0 rz 0.01 deg; joints [32.487, -41.052, 99.085, -143.312, 64.067, 162.939]
  MoveL 7903 to (-264.11, 138.12, -64.5) mm, rotated rx 180 ry 0 rz 0.01 deg; joints [32.513, -41.147, 99.292, -143.317, 64.166, 163.001]
  MoveL 7904 to (-263.74, 138, -64.5) mm, rotated rx 180 ry 0 rz 0.01 deg; joints [32.517, -41.163, 99.328, -143.319, 64.183, 163.012]
  MoveL 7905 to (-260.65, 136.81, -64.5) mm, rotated rx -180 ry 0 rz 0.01 deg; joints [32.541, -41.306, 99.642, -143.343, 64.328, 163.115]
  MoveL 7906 to (-260.33, 136.67, -64.5) mm, rotated rx -180 ry 0 rz 0.01 deg; joints [32.543, -41.321, 99.675, -143.346, 64.343, 163.126]
  MoveL 7907 to (-258.3, 135.64, -64.5) mm, rotated rx 180 ry 0 rz 0.01 deg; joints [32.551, -41.42, 99.893, -143.371, 64.441, 163.2]
  MoveL 7908 to (-258.15, 135.55, -64.5) mm, rotated rx 180 ry 0 rz 0.01 deg; joints [32.552, -41.428, 99.91, -143.373, 64.448, 163.206]
  MoveL 7909 to (-222.39, 114.98, -64.5) mm, rotated rx -180 ry 0 rz 0.01 deg; joints [32.624, -43.186, 103.807, -143.88, 66.192, 164.569]
  MoveL 7910 to (-221.74, 114.49, -64.5) mm, rotated rx 180 ry 0 rz 0.01 deg; joints [32.622, -43.22, 103.882, -143.893, 66.225, 164.597]
  MoveL 7911 to (-220.98, 113.77, -64.5) mm, rotated rx 180 ry 0 rz 0.01 deg; joints [32.614, -43.263, 103.978, -143.915, 66.265, 164.635]
  MoveC 7912 to (-220.64, 113.39, -64.5) mm, rotated rx 180 ry 0 rz 0.01 deg; joints [32.609, -43.283, 104.023, -143.927, 66.284, 164.653] to (-220.37, 112.97, -64.5) mm, rotated rx 180 ry 0 rz 0.01 deg; joints [32.601, -43.302, 104.066, -143.941, 66.301, 164.672]
  MoveL 7913 to (-219.87, 112.08, -64.5) mm, rotated rx -180 ry 0 rz 0.01 deg; joints [32.583, -43.339, 104.148, -143.972, 66.333, 164.709]
  MoveC 7914 to (-219.65, 111.61, -64.5) mm, rotated rx 180 ry 0 rz 0.01 deg; joints [32.572, -43.357, 104.189, -143.989, 66.348, 164.728] to (-219.51, 111.11, -64.5) mm, rotated rx 180 ry 0 rz 0.01 deg; joints [32.559, -43.373, 104.225, -144.008, 66.361, 164.747]
  MoveL 7915 to (-219.29, 110.02, -64.5) mm, rotated rx 180 ry 0 rz 0.01 deg; joints [32.528, -43.404, 104.297, -144.051, 66.384, 164.786]
  MoveC 7916 to (-219.22, 109.49, -64.5) mm, rotated rx -180 ry 0 rz 0.01 deg; joints [32.512, -43.418, 104.328, -144.072, 66.394, 164.804] to (-219.25, 108.95, -64.5) mm, rotated rx 180 ry 0 rz 0.01 deg; joints [32.494, -43.429, 104.353, -144.094, 66.401, 164.821]
  MoveL 7917 to (-219.37, 107.86, -64.5) mm, rotated rx -180 ry 0 rz 0.01 deg; joints [32.456, -43.448, 104.397, -144.14, 66.41, 164.853]
  MoveC 7918 to (-219.49, 107.32, -64.5) mm, rotated rx 180 ry 0 rz 0.01 deg; joints [32.437, -43.456, 104.416, -144.164, 66.413, 164.868] to (-219.68, 106.8, -64.5) mm, rotated rx 180 ry 0 rz 0.01 deg; joints [32.416, -43.46, 104.426, -144.187, 66.412, 164.881]
  MoveL 7919 to (-220.19, 105.74, -64.5) mm, rotated rx 180 ry 0 rz 0.01 deg; joints [32.371, -43.465, 104.439, -144.236, 66.406, 164.905]
  MoveC 7920 to (-220.45, 105.29, -64.5) mm, rotated rx -180 ry 0 rz 0.01 deg; joints [32.351, -43.465, 104.44, -144.258, 66.401, 164.915] to (-220.79, 104.88, -64.5) mm, rotated rx 180 ry 0 rz 0.01 deg; joints [32.331, -43.462, 104.435, -144.278, 66.393, 164.922]
  MoveL 7921 to (-221.46, 104.16, -64.5) mm, rotated rx 180 ry 0 rz 0.01 deg; joints [32.294, -43.453, 104.417, -144.315, 66.375, 164.932]
  MoveL 7922 to (-222.23, 103.56, -64.5) mm, rotated rx 180 ry 0 rz 0.01 deg; joints [32.258, -43.439, 104.387, -144.347, 66.352, 164.937]
  MoveL 7923 to (-337.67, 36.98, -64.5) mm, rotated rx -180 ry 0 rz 0.01 deg; joints [27.92, -40.489, 98.046, -148.057, 62.303, 164.89]
  MoveL 7924 to (-329.75, 23.29, -64.5) mm, rotated rx -180 ry 0 rz 0.01 deg; joints [27.609, -41.074, 99.346, -148.589, 62.825, 165.472]
  MoveL 7925 to (-214.41, 89.96, -64.5) mm, rotated rx -180 ry 0 rz 0.01 deg; joints [31.974, -44.004, 105.662, -144.823, 66.853, 165.507]
  MoveL 7926 to (-213.53, 90.32, -64.5) mm, rotated rx -180 ry 0 rz 0.01 deg; joints [32.004, -44.027, 105.713, -144.798, 66.883, 165.512]
  MoveL 7927 to (-212.57, 90.56, -64.5) mm, rotated rx 180 ry 0 rz 0.01 deg; joints [32.032, -44.056, 105.776, -144.778, 66.919, 165.522]
  MoveL 7928 to (-211.59, 90.65, -64.5) mm, rotated rx 180 ry 0 rz 0.01 deg; joints [32.055, -44.088, 105.848, -144.763, 66.958, 165.536]
  MoveL 7929 to (-210.55, 90.6, -64.5) mm, rotated rx 180 ry 0 rz 0.01 deg; joints [32.075, -44.125, 105.931, -144.754, 67, 165.557]
  MoveL 7930 to (-209.59, 90.41, -64.5) mm, rotated rx 180 ry 0 rz 0.01 deg; joints [32.088, -44.163, 106.014, -144.751, 67.041, 165.58]
  MoveL 7931 to (-208.69, 90.09, -64.5) mm, rotated rx 180 ry 0 rz 0.01 deg; joints [32.096, -44.201, 106.1, -144.754, 67.082, 165.606]
  MoveC 7932 to (-208.22, 89.88, -64.5) mm, rotated rx -180 ry 0 rz 0.01 deg; joints [32.099, -44.222, 106.146, -144.757, 67.104, 165.621] to (-207.79, 89.61, -64.5) mm, rotated rx 180 ry 0 rz 0.01 deg; joints [32.099, -44.242, 106.192, -144.764, 67.125, 165.637]
  MoveL 7933 to (-206.89, 88.94, -64.5) mm, rotated rx -180 ry 0 rz 0.01 deg; joints [32.096, -44.288, 106.295, -144.781, 67.17, 165.674]
  MoveC 7934 to (-206.47, 88.57, -64.5) mm, rotated rx 180 ry 0 rz 0.01 deg; joints [32.092, -44.31, 106.345, -144.792, 67.192, 165.693] to (-206.12, 88.14, -64.5) mm, rotated rx 180 ry 0 rz 0.01 deg; joints [32.085, -44.331, 106.392, -144.805, 67.212, 165.713]
  MoveL 7935 to (-205.48, 87.2, -64.5) mm, rotated rx 180 ry 0 rz 0.01 deg; joints [32.067, -44.373, 106.488, -144.837, 67.251, 165.753]
  MoveC 7936 to (-205.22, 86.74, -64.5) mm, rotated rx 180 ry 0 rz 0.01 deg; joints [32.058, -44.392, 106.53, -144.852, 67.267, 165.772] to (-205.03, 86.25, -64.5) mm, rotated rx 180 ry 0 rz 0.01 deg; joints [32.046, -44.409, 106.568, -144.87, 67.282, 165.79]
  MoveL 7937 to (-204.74, 85.29, -64.5) mm, rotated rx 180 ry 0 rz 0.01 deg; joints [32.02, -44.439, 106.637, -144.907, 67.306, 165.825]
  MoveL 7938 to (-204.6, 84.32, -64.5) mm, rotated rx 180 ry 0 rz 0.01 deg; joints [31.99, -44.464, 106.694, -144.945, 67.325, 165.858]
  MoveL 7939 to (-204.63, 42.24, -64.5) mm, rotated rx -180 ry 0 rz 0.01 deg; joints [30.575, -45.306, 108.66, -146.685, 67.89, 167.119]
  MoveL 7940 to (-204.64, 41.91, -64.5) mm, rotated rx 180 ry 0 rz 0.01 deg; joints [30.563, -45.312, 108.673, -146.698, 67.894, 167.128]
  MoveL 7941 to (-204.93, 39.01, -64.5) mm, rotated rx -180 ry 0 rz 0.01 deg; joints [30.458, -45.358, 108.783, -146.822, 67.921, 167.208]
  MoveL 7942 to (-204.98, 38.69, -64.5) mm, rotated rx -180 ry 0 rz 0.01 deg; joints [30.447, -45.363, 108.793, -146.836, 67.923, 167.216]
  MoveL 7943 to (-205.54, 35.79, -64.5) mm, rotated rx 180 ry 0 rz 0.01 deg; joints [30.336, -45.399, 108.881, -146.963, 67.939, 167.291]
  MoveL 7944 to (-205.63, 35.43, -64.5) mm, rotated rx 180 ry 0 rz 0.01 deg; joints [30.322, -45.403, 108.89, -146.979, 67.94, 167.3]
  MoveL 7945 to (-206.08, 33.98, -64.5) mm, rotated rx 180 ry 0 rz 0.01 deg; joints [30.263, -45.415, 108.92, -147.045, 67.941, 167.334]
  MoveL 7946 to (-206.22, 33.63, -64.5) mm, rotated rx 180 ry 0 rz 0.01 deg; joints [30.248, -45.417, 108.926, -147.061, 67.94, 167.342]
  MoveL 7947 to (-207.11, 31.59, -64.5) mm, rotated rx 180 ry 0 rz 0.01 deg; joints [30.16, -45.425, 108.949, -147.156, 67.931, 167.386]
  MoveL 7948 to (-207.43, 31.01, -64.5) mm, rotated rx 180 ry 0 rz 0.01 deg; joints [30.134, -45.425, 108.949, -147.184, 67.926, 167.398]
  MoveL 7949 to (-208.44, 29.57, -64.5) mm, rotated rx 180 ry 0 rz 0.01 deg; joints [30.064, -45.418, 108.936, -147.255, 67.904, 167.422]
  MoveL 7950 to (-208.78, 29.16, -64.5) mm, rotated rx -180 ry 0 rz 0.01 deg; joints [30.044, -45.414, 108.928, -147.276, 67.895, 167.428]
  MoveL 7951 to (-209.55, 28.36, -64.5) mm, rotated rx 180 ry 0 rz 0.01 deg; joints [30.001, -45.403, 108.904, -147.318, 67.875, 167.438]
  MoveL 7952 to (-210.05, 27.93, -64.5) mm, rotated rx 180 ry 0 rz 0.01 deg; joints [29.976, -45.393, 108.884, -147.342, 67.86, 167.442]
  MoveL 7953 to (-211.66, 26.81, -64.5) mm, rotated rx 180 ry 0 rz 0.01 deg; joints [29.906, -45.359, 108.809, -147.407, 67.809, 167.447]
  MoveL 7954 to (-212.2, 26.5, -64.5) mm, rotated rx 180 ry 0 rz 0.01 deg; joints [29.884, -45.346, 108.781, -147.426, 67.791, 167.447]
  MoveL 7955 to (-336.13, -29.42, -64.5) mm, rotated rx 180 ry 0 rz 0.01 deg; joints [25.746, -41.811, 101.064, -150.859, 63.185, 166.964]
  MoveL 7956 to (-336.25, -29.48, -64.5) mm, rotated rx 180 ry 0 rz 0.01 deg; joints [25.742, -41.807, 101.055, -150.862, 63.18, 166.963]
  MoveL 7957 to (-339.16, -30.64, -64.5) mm, rotated rx 180 ry 0 rz 0.01 deg; joints [25.656, -41.714, 100.854, -150.93, 63.064, 166.947]
  MoveL 7958 to (-339.41, -30.73, -64.5) mm, rotated rx 180 ry 0 rz 0.01 deg; joints [25.648, -41.706, 100.837, -150.935, 63.053, 166.946]
  MoveL 7959 to (-341.1, -31.27, -64.5) mm, rotated rx 180 ry 0 rz 0.01 deg; joints [25.603, -41.649, 100.713, -150.968, 62.984, 166.932]
  MoveL 7960 to (-52.41, -31.27, -64.5) mm, rotated rx 180 ry 0 rz 0.01 deg; joints [31.21, -51.458, 122.995, -147.527, 74.898, 171.59]
  MoveL 7961 to (-54.11, -30.73, -64.5) mm, rotated rx -180 ry 0 rz 0.01 deg; joints [31.191, -51.399, 122.854, -147.534, 74.825, 171.549]
  MoveL 7962 to (-54.38, -30.64, -64.5) mm, rotated rx -180 ry 0 rz 0.01 deg; joints [31.188, -51.39, 122.831, -147.535, 74.814, 171.543]
  MoveL 7963 to (-58.15, -29.08, -64.5) mm, rotated rx -180 ry 0 rz 0.01 deg; joints [31.16, -51.254, 122.503, -147.535, 74.646, 171.443]
  MoveL 7964 to (-58.26, -29.04, -64.5) mm, rotated rx -180 ry 0 rz 0.01 deg; joints [31.159, -51.25, 122.493, -147.535, 74.642, 171.441]
  MoveL 7965 to (-181.53, 26.63, -64.5) mm, rotated rx 180 ry 0 rz 0.01 deg; joints [30.507, -46.39, 111.128, -147.055, 69.033, 167.959]
  MoveL 7966 to (-182.15, 26.99, -64.5) mm, rotated rx 180 ry 0 rz 0.01 deg; joints [30.507, -46.362, 111.064, -147.047, 69.003, 167.938]
  MoveL 7967 to (-183.79, 28.21, -64.5) mm, rotated rx 180 ry 0 rz 0.01 deg; joints [30.515, -46.284, 110.886, -147.017, 68.921, 167.877]
  MoveL 7968 to (-184.36, 28.74, -64.5) mm, rotated rx -180 ry 0 rz 0.01 deg; joints [30.522, -46.255, 110.819, -147.002, 68.891, 167.852]
  MoveL 7969 to (-185.34, 29.91, -64.5) mm, rotated rx -180 ry 0 rz 0.01 deg; joints [30.542, -46.2, 110.693, -146.966, 68.836, 167.802]
  MoveL 7970 to (-185.67, 30.38, -64.5) mm, rotated rx -180 ry 0 rz 0.01 deg; joints [30.552, -46.18, 110.647, -146.95, 68.816, 167.783]
  MoveL 7971 to (-186.43, 31.68, -64.5) mm, rotated rx 180 ry 0 rz 0.01 deg; joints [30.582, -46.129, 110.53, -146.905, 68.768, 167.733]
  MoveL 7972 to (-186.62, 32.06, -64.5) mm, rotated rx -180 ry 0 rz 0.01 deg; joints [30.591, -46.116, 110.499, -146.892, 68.755, 167.719]
  MoveL 7973 to (-187.31, 33.65, -64.5) mm, rotated rx -180 ry 0 rz 0.01 deg; joints [30.632, -46.063, 110.375, -146.834, 68.706, 167.662]
  MoveL 7974 to (-187.43, 33.98, -64.5) mm, rotated rx -180 ry 0 rz 0.01 deg; joints [30.641, -46.052, 110.351, -146.822, 68.697, 167.65]
  MoveL 7975 to (-187.88, 35.43, -64.5) mm, rotated rx -180 ry 0 rz 0.01 deg; joints [30.682, -46.009, 110.251, -146.767, 68.659, 167.601]
  MoveL 7976 to (-187.97, 35.79, -64.5) mm, rotated rx -180 ry 0 rz 0.01 deg; joints [30.692, -45.999, 110.228, -146.754, 68.65, 167.589]
  MoveL 7977 to (-188.54, 38.69, -64.5) mm, rotated rx -180 ry 0 rz 0.01 deg; joints [30.781, -45.925, 110.054, -146.64, 68.588, 167.496]
  MoveL 7978 to (-188.58, 39.01, -64.5) mm, rotated rx -180 ry 0 rz 0.01 deg; joints [30.79, -45.917, 110.036, -146.627, 68.582, 167.486]
  MoveL 7979 to (-188.87, 41.91, -64.5) mm, rotated rx 180 ry 0 rz 0.01 deg; joints [30.884, -45.852, 109.883, -146.511, 68.532, 167.397]
  MoveL 7980 to (-188.88, 42.24, -64.5) mm, rotated rx 180 ry 0 rz 0.01 deg; joints [30.895, -45.845, 109.867, -146.497, 68.527, 167.388]
  MoveL 7981 to (-188.91, 84.32, -64.5) mm, rotated rx 180 ry 0 rz 0.01 deg; joints [32.318, -45.003, 107.897, -144.761, 67.954, 166.137]
  MoveL 7982 to (-188.77, 85.29, -64.5) mm, rotated rx -180 ry 0 rz 0.01 deg; joints [32.353, -44.988, 107.861, -144.719, 67.946, 166.11]
  MoveL 7983 to (-188.48, 86.25, -64.5) mm, rotated rx 180 ry 0 rz 0.01 deg; joints [32.391, -44.978, 107.836, -144.676, 67.945, 166.085]
  MoveC 7984 to (-188.3, 86.74, -64.5) mm, rotated rx 180 ry 0 rz 0.01 deg; joints [32.412, -44.974, 107.827, -144.653, 67.945, 166.074] to (-188.03, 87.2, -64.5) mm, rotated rx -180 ry 0 rz 0.01 deg; joints [32.432, -44.974, 107.825, -144.632, 67.95, 166.064]
  MoveL 7985 to (-187.39, 88.14, -64.5) mm, rotated rx 180 ry 0 rz 0.01 deg; joints [32.477, -44.976, 107.829, -144.585, 67.962, 166.047]
  MoveL 7986 to (-186.93, 88.67, -64.5) mm, rotated rx -180 ry 0 rz 0.01 deg; joints [32.505, -44.981, 107.837, -144.558, 67.973, 166.039]
  MoveL 7987 to (-186.72, 88.88, -64.5) mm, rotated rx 180 ry 0 rz 0.01 deg; joints [32.516, -44.984, 107.844, -144.547, 67.979, 166.036]
  MoveL 7988 to (-186.19, 89.29, -64.5) mm, rotated rx -180 ry 0 rz 0.01 deg; joints [32.541, -44.993, 107.864, -144.523, 67.994, 166.033]
  MoveL 7989 to (-185.27, 89.87, -64.5) mm, rotated rx -180 ry 0 rz 0.01 deg; joints [32.579, -45.012, 107.906, -144.488, 68.023, 166.032]
  MoveC 7990 to (-184.81, 90.11, -64.5) mm, rotated rx -180 ry 0 rz 0.01 deg; joints [32.597, -45.023, 107.929, -144.473, 68.038, 166.033] to (-184.32, 90.28, -64.5) mm, rotated rx 180 ry 0 rz 0.01 deg; joints [32.614, -45.036, 107.958, -144.46, 68.055, 166.036]
  MoveL 7991 to (-183.29, 90.55, -64.5) mm, rotated rx -180 ry 0 rz 0.01 deg; joints [32.644, -45.066, 108.023, -144.436, 68.092, 166.046]
  MoveC 7992 to (-182.79, 90.64, -64.5) mm, rotated rx -180 ry 0 rz 0.01 deg; joints [32.658, -45.081, 108.057, -144.426, 68.111, 166.052] to (-182.28, 90.65, -64.5) mm, rotated rx 180 ry 0 rz 0.01 deg; joints [32.669, -45.098, 108.095, -144.42, 68.131, 166.061]
  MoveL 7993 to (-181.24, 90.6, -64.5) mm, rotated rx 180 ry 0 rz 0.01 deg; joints [32.69, -45.134, 108.177, -144.409, 68.173, 166.081]
  MoveC 7994 to (-180.73, 90.53, -64.5) mm, rotated rx -180 ry 0 rz 0.01 deg; joints [32.698, -45.153, 108.218, -144.405, 68.194, 166.092] to (-180.24, 90.4, -64.5) mm, rotated rx -180 ry 0 rz 0.01 deg; joints [32.704, -45.172, 108.262, -144.405, 68.215, 166.105]
  MoveL 7995 to (-179.27, 90.04, -64.5) mm, rotated rx 180 ry 0 rz 0.01 deg; joints [32.713, -45.213, 108.353, -144.407, 68.259, 166.133]
  MoveL 7996 to (-178.74, 89.79, -64.5) mm, rotated rx -180 ry 0 rz 0.01 deg; joints [32.716, -45.236, 108.404, -144.411, 68.283, 166.15]
  MoveL 7997 to (-63.76, 23.29, -64.5) mm, rotated rx 180 ry 0 rz 0.01 deg; joints [32.986, -50.176, 119.829, -145.42, 73.654, 169.998]
  MoveL 7998 to (-55.84, 36.98, -64.5) mm, rotated rx 180 ry 0 rz 0.01 deg; joints [33.674, -50.158, 119.755, -144.708, 73.745, 169.76]
  MoveL 7999 to (-171.28, 103.56, -64.5) mm, rotated rx 180 ry 0 rz 0.01 deg; joints [33.333, -45.198, 108.293, -143.753, 68.387, 165.861]
  MoveL 8000 to (-172.05, 104.16, -64.5) mm, rotated rx -180 ry 0 rz 0.01 deg; joints [33.337, -45.16, 108.206, -143.739, 68.349, 165.828]
  MoveL 8001 to (-172.73, 104.88, -64.5) mm, rotated rx -180 ry 0 rz 0.01 deg; joints [33.345, -45.122, 108.12, -143.718, 68.312, 165.794]
  MoveC 8002 to (-173.06, 105.29, -64.5) mm, rotated rx -180 ry 0 rz 0.01 deg; joints [33.352, -45.102, 108.075, -143.705, 68.294, 165.776] to (-173.32, 105.74, -64.5) mm, rotated rx 180 ry 0 rz 0.01 deg; joints [33.361, -45.083, 108.033, -143.69, 68.277, 165.757]
  MoveL 8003 to (-173.83, 106.8, -64.5) mm, rotated rx 180 ry 0 rz 0.01 deg; joints [33.385, -45.044, 107.942, -143.654, 68.242, 165.715]
  MoveC 8004 to (-174.03, 107.32, -64.5) mm, rotated rx -180 ry 0 rz 0.01 deg; joints [33.398, -45.026, 107.902, -143.635, 68.227, 165.695] to (-174.14, 107.86, -64.5) mm, rotated rx 180 ry 0 rz 0.01 deg; joints [33.413, -45.011, 107.867, -143.614, 68.216, 165.677]
  MoveL 8005 to (-174.27, 108.95, -64.5) mm, rotated rx -180 ry 0 rz 0.01 deg; joints [33.446, -44.983, 107.803, -143.571, 68.195, 165.64]
  MoveC 8006 to (-174.29, 109.49, -64.5) mm, rotated rx -180 ry 0 rz 0.01 deg; joints [33.463, -44.971, 107.775, -143.55, 68.187, 165.623] to (-174.22, 110.02, -64.5) mm, rotated rx -180 ry 0 rz 0.01 deg; joints [33.482, -44.962, 107.753, -143.527, 68.182, 165.608]
  MoveL 8007 to (-174, 111.11, -64.5) mm, rotated rx -180 ry 0 rz 0.01 deg; joints [33.523, -44.946, 107.715, -143.48, 68.176, 165.578]
  MoveC 8008 to (-173.86, 111.61, -64.5) mm, rotated rx -180 ry 0 rz 0.01 deg; joints [33.542, -44.94, 107.701, -143.458, 68.175, 165.565] to (-173.64, 112.08, -64.5) mm, rotated rx 180 ry 0 rz 0.01 deg; joints [33.563, -44.937, 107.694, -143.436, 68.177, 165.554]
  MoveL 8009 to (-173.15, 112.97, -64.5) mm, rotated rx 180 ry 0 rz 0.01 deg; joints [33.602, -44.935, 107.687, -143.393, 68.184, 165.535]
  MoveC 8010 to (-172.87, 113.39, -64.5) mm, rotated rx -180 ry 0 rz 0.01 deg; joints [33.622, -44.935, 107.687, -143.373, 68.189, 165.527] to (-172.53, 113.77, -64.5) mm, rotated rx -180 ry 0 rz 0.01 deg; joints [33.642, -44.938, 107.694, -143.353, 68.197, 165.522]
  MoveL 8011 to (-171.78, 114.49, -64.5) mm, rotated rx -180 ry 0 rz 0.01 deg; joints [33.682, -44.948, 107.714, -143.314, 68.217, 165.513]
  MoveL 8012 to (-171.12, 114.98, -64.5) mm, rotated rx -180 ry 0 rz 0.01 deg; joints [33.712, -44.96, 107.739, -143.286, 68.235, 165.509]
  MoveL 8013 to (-134.69, 135.94, -64.5) mm, rotated rx -180 ry 0 rz 0.01 deg; joints [35.214, -45.708, 109.372, -141.945, 69.348, 165.508]
  MoveL 8014 to (-134.37, 136.1, -64.5) mm, rotated rx -180 ry 0 rz 0.01 deg; joints [35.226, -45.715, 109.386, -141.934, 69.358, 165.509]
  MoveL 8015 to (-131.37, 137.43, -64.5) mm, rotated rx 180 ry 0 rz 0.01 deg; joints [35.338, -45.783, 109.536, -141.838, 69.453, 165.521]
  MoveL 8016 to (-131.12, 137.53, -64.5) mm, rotated rx 180 ry 0 rz 0.01 deg; joints [35.348, -45.789, 109.55, -141.83, 69.462, 165.522]
  MoveL 8017 to (-129.67, 138.04, -64.5) mm, rotated rx -180 ry 0 rz 0.01 deg; joints [35.398, -45.825, 109.629, -141.789, 69.509, 165.533]
  MoveL 8018 to (-129.41, 138.12, -64.5) mm, rotated rx 180 ry 0 rz 0.01 deg; joints [35.406, -45.832, 109.644, -141.782, 69.518, 165.535]
  MoveL 8019 to (-127.23, 138.69, -64.5) mm, rotated rx 180 ry 0 rz 0.01 deg; joints [35.475, -45.889, 109.772, -141.727, 69.592, 165.556]
  MoveL 8020 to (-126.74, 138.78, -64.5) mm, rotated rx 180 ry 0 rz 0.01 deg; joints [35.489, -45.903, 109.803, -141.717, 69.61, 165.562]
  MoveL 8021 to (-124.2, 139.05, -64.5) mm, rotated rx 180 ry 0 rz 0.01 deg; joints [35.558, -45.979, 109.972, -141.668, 69.702, 165.599]
  MoveL 8022 to (-123.56, 139.06, -64.5) mm, rotated rx 180 ry 0 rz 0.01 deg; joints [35.573, -45.999, 110.018, -141.658, 69.726, 165.61]
  MoveL 8023 to (-122.11, 138.94, -64.5) mm, rotated rx 180 ry 0 rz 0.01 deg; joints [35.603, -46.049, 110.129, -141.642, 69.782, 165.64]
  MoveL 8024 to (-121.51, 138.84, -64.5) mm, rotated rx 180 ry 0 rz 0.01 deg; joints [35.613, -46.07, 110.177, -141.637, 69.806, 165.654]
  MoveL 8025 to (-120.06, 138.45, -64.5) mm, rotated rx -180 ry 0 rz 0.01 deg; joints [35.635, -46.125, 110.302, -141.631, 69.866, 165.692]
  MoveL 8026 to (-119.49, 138.24, -64.5) mm, rotated rx 180 ry 0 rz 0.01 deg; joints [35.641, -46.148, 110.353, -141.631, 69.891, 165.709]
  MoveL 8027 to (-118.01, 137.54, -64.5) mm, rotated rx -180 ry 0 rz 0.01 deg; joints [35.653, -46.211, 110.496, -141.637, 69.956, 165.757]
  MoveL 8028 to (-117.48, 137.23, -64.5) mm, rotated rx 180 ry 0 rz 0.01 deg; joints [35.655, -46.234, 110.55, -141.642, 69.981, 165.776]
  MoveL 8029 to (-7.3, 58.05, -64.5) mm, rotated rx -180 ry 0 rz 0.01 deg; joints [35.65, -51.159, 122.062, -142.912, 75.193, 170.001]
  MoveL 8030 to (-7.2, 57.97, -64.5) mm, rotated rx -180 ry 0 rz 0.01 deg; joints [35.65, -51.163, 122.073, -142.913, 75.198, 170.005]
  MoveL 8031 to (-4.57, 55.92, -64.5) mm, rotated rx -180 ry 0 rz 0.01 deg; joints [35.644, -51.275, 122.344, -142.945, 75.324, 170.106]
  MoveL 8032 to (-4.36, 55.74, -64.5) mm, rotated rx 180 ry 0 rz 0.01 deg; joints [35.643, -51.285, 122.367, -142.948, 75.334, 170.114]
  MoveL 8033 to (-1.46, 53.05, -64.5) mm, rotated rx 180 ry 0 rz 0.01 deg; joints [35.621, -51.417, 122.687, -143, 75.48, 170.237]
  MoveL 8034 to (-1.21, 52.8, -64.5) mm, rotated rx -180 ry 0 rz 0.01 deg; joints [35.618, -51.429, 122.716, -143.005, 75.493, 170.248]
  MoveL 8035 to (2.28, 48.82, -64.5) mm, rotated rx 180 ry 0 rz 0.01 deg; joints [35.564, -51.601, 123.135, -143.098, 75.68, 170.416]
  MoveL 8036 to (2.64, 48.33, -64.5) mm, rotated rx 180 ry 0 rz 0.01 deg; joints [35.556, -51.62, 123.182, -143.111, 75.701, 170.435]
  MoveL 8037 to (4.95, 44.47, -64.5) mm, rotated rx 180 ry 0 rz 0.01 deg; joints [35.475, -51.756, 123.517, -143.223, 75.844, 170.579]
  MoveL 8038 to (4.98, 44.43, -64.5) mm, rotated rx 180 ry 0 rz 0.01 deg; joints [35.474, -51.757, 123.52, -143.224, 75.846, 170.581]
  MoveL 8039 to (8.27, 38.74, -64.5) mm, rotated rx -180 ry 0 rz 0.01 deg; joints [35.351, -51.954, 124.004, -143.392, 76.054, 170.79]
  MoveL 8040 to (8.49, 38.28, -64.5) mm, rotated rx -180 ry 0 rz 0.01 deg; joints [35.339, -51.968, 124.04, -143.407, 76.069, 170.806]
  MoveL 8041 to (9.3, 36.22, -64.5) mm, rotated rx 180 ry 0 rz 0.01 deg; joints [35.284, -52.028, 124.19, -143.476, 76.131, 170.875]
  MoveL 8042 to (9.44, 35.74, -64.5) mm, rotated rx 180 ry 0 rz 0.01 deg; joints [35.27, -52.041, 124.222, -143.493, 76.144, 170.89]
  MoveL 8043 to (10.27, 32.11, -64.5) mm, rotated rx 180 ry 0 rz 0.01 deg; joints [35.157, -52.13, 124.445, -143.627, 76.231, 171]
  MoveL 8044 to (10.27, 334.35, -64.5) mm, rotated rx -180 ry 0 rz 0.01 deg; joints [44.94, -45.196, 107.88, -131.889, 71.632, 161.403]
  MoveL 8045 to (10.07, 335.56, -64.5) mm, rotated rx 180 ry 0 rz 0.01 deg; joints [44.968, -45.157, 107.79, -131.849, 71.608, 161.354]
  MoveL 8046 to (9.9, 336.02, -64.5) mm, rotated rx 180 ry 0 rz 0.01 deg; joints [44.976, -45.139, 107.75, -131.835, 71.596, 161.334]
  MoveL 8047 to (9.66, 336.38, -64.5) mm, rotated rx 180 ry 0 rz 0.01 deg; joints [44.98, -45.122, 107.712, -131.827, 71.583, 161.316]
  MoveL 8048 to (7.37, 338.63, -64.5) mm, rotated rx -180 ry 0 rz 0.01 deg; joints [44.979, -44.994, 107.422, -131.787, 71.475, 161.19]
  MoveL 8049 to (7.07, 338.84, -64.5) mm, rotated rx -180 ry 0 rz 0.01 deg; joints [44.976, -44.979, 107.389, -131.786, 71.462, 161.176]
  MoveL 8050 to (6.8, 338.95, -64.5) mm, rotated rx 180 ry 0 rz 0.01 deg; joints [44.972, -44.968, 107.365, -131.786, 71.451, 161.167]
  MoveL 8051 to (5.94, 339.15, -64.5) mm, rotated rx 180 ry 0 rz 0.01 deg; joints [44.953, -44.938, 107.297, -131.795, 71.42, 161.144]
  MoveL 8052 to (4.87, 339.21, -64.5) mm, rotated rx 180 ry 0 rz 0.01 deg; joints [44.925, -44.905, 107.224, -131.813, 71.384, 161.122]
  MoveL 8053 to (-180.11, 339.2, -64.5) mm, rotated rx -180 ry 0 rz 0.01 deg; joints [40.236, -38.946, 94.19, -134.422, 64.774, 157.353]
  MoveL 8054 to (-179.93, 339.18, -64.5) mm, rotated rx 180 ry 0 rz 0.01 deg; joints [40.239, -38.953, 94.206, -134.421, 64.782, 157.358]
  MoveL 8055 to (-179.33, 339.03, -64.5) mm, rotated rx -180 ry 0 rz 0.01 deg; joints [40.249, -38.979, 94.262, -134.422, 64.807, 157.377]
  MoveL 8056 to (-178.24, 338.66, -64.5) mm, rotated rx 180 ry 0 rz 0.01 deg; joints [40.264, -39.029, 94.371, -134.426, 64.854, 157.417]
  MoveL 8057 to (-177.87, 338.5, -64.5) mm, rotated rx 180 ry 0 rz 0.01 deg; joints [40.268, -39.047, 94.41, -134.429, 64.87, 157.431]
  MoveL 8058 to (-167.35, 333.4, -64.5) mm, rotated rx 180 ry 0 rz 0.01 deg; joints [40.374, -39.571, 95.549, -134.526, 65.344, 157.869]
  MoveL 8059 to (-166.81, 333.08, -64.5) mm, rotated rx 180 ry 0 rz 0.01 deg; joints [40.377, -39.6, 95.611, -134.533, 65.368, 157.894]
  MoveL 8060 to (-165.36, 332.01, -64.5) mm, rotated rx -180 ry 0 rz 0.01 deg; joints [40.382, -39.682, 95.791, -134.561, 65.439, 157.969]
  MoveL 8061 to (-165.06, 331.76, -64.5) mm, rotated rx 180 ry 0 rz 0.01 deg; joints [40.382, -39.7, 95.829, -134.567, 65.453, 157.985]
  MoveL 8062 to (-157.16, 324.39, -64.5) mm, rotated rx -180 ry 0 rz 0.01 deg; joints [40.364, -40.189, 96.901, -134.773, 65.855, 158.447]
  MoveL 8063 to (-156.79, 323.99, -64.5) mm, rotated rx 180 ry 0 rz 0.01 deg; joints [40.361, -40.214, 96.955, -134.785, 65.875, 158.471]
  MoveL 8064 to (-155.39, 322.17, -64.5) mm, rotated rx -180 ry 0 rz 0.01 deg; joints [40.344, -40.315, 97.176, -134.84, 65.953, 158.572]
  MoveL 8065 to (-155.13, 321.78, -64.5) mm, rotated rx -180 ry 0 rz 0.01 deg; joints [40.339, -40.335, 97.22, -134.853, 65.968, 158.592]
  MoveL 8066 to (-149.95, 312.72, -64.5) mm, rotated rx -180 ry 0 rz 0.01 deg; joints [40.209, -40.772, 98.183, -135.149, 66.29, 159.054]
  MoveL 8067 to (-149.71, 312.2, -64.5) mm, rotated rx 180 ry 0 rz 0.01 deg; joints [40.2, -40.795, 98.233, -135.167, 66.306, 159.079]
  MoveL 8068 to (-148.51, 308.94, -64.5) mm, rotated rx 180 ry 0 rz 0.01 deg; joints [40.136, -40.928, 98.527, -135.28, 66.397, 159.229]
  MoveL 8069 to (-148.44, 308.73, -64.5) mm, rotated rx 180 ry 0 rz 0.01 deg; joints [40.132, -40.936, 98.546, -135.288, 66.402, 159.239]
  MoveL 8070 to (-147.59, 305.82, -64.5) mm, rotated rx -180 ry 0 rz 0.01 deg; joints [40.07, -41.046, 98.791, -135.391, 66.475, 159.367]
  MoveL 8071 to (-147.53, 305.6, -64.5) mm, rotated rx 180 ry 0 rz 0.01 deg; joints [40.066, -41.055, 98.809, -135.399, 66.48, 159.377]
  MoveL 8072 to (-146.88, 302.7, -64.5) mm, rotated rx -180 ry 0 rz 0.01 deg; joints [39.999, -41.158, 99.038, -135.505, 66.545, 159.501]
  MoveL 8073 to (-146.84, 302.44, -64.5) mm, rotated rx -180 ry 0 rz 0.01 deg; joints [39.992, -41.166, 99.058, -135.515, 66.55, 159.512]
  MoveL 8074 to (-146.43, 299.54, -64.5) mm, rotated rx 180 ry 0 rz 0.01 deg; joints [39.92, -41.261, 99.268, -135.624, 66.606, 159.63]
  MoveL 8075 to (-146.41, 299.4, -64.5) mm, rotated rx 180 ry 0 rz 0.01 deg; joints [39.916, -41.265, 99.278, -135.629, 66.609, 159.636]
  MoveL 8076 to (-132.85, 163.73, -64.5) mm, rotated rx -180 ry 0 rz 0.01 deg; joints [36.151, -45.144, 108.056, -140.804, 69.025, 164.655]
  MoveL 8077 to (-132.86, 162.99, -64.5) mm, rotated rx -180 ry 0 rz 0.01 deg; joints [36.127, -45.161, 108.095, -140.834, 69.035, 164.679]
  MoveL 8078 to (-133.12, 160.81, -64.5) mm, rotated rx 180 ry 0 rz 0.01 deg; joints [36.052, -45.202, 108.191, -140.925, 69.056, 164.744]
  MoveL 8079 to (-133.32, 160.02, -64.5) mm, rotated rx -180 ry 0 rz 0.01 deg; joints [36.022, -45.214, 108.219, -140.959, 69.06, 164.766]
  MoveL 8080 to (-133.87, 158.57, -64.5) mm, rotated rx 180 ry 0 rz 0.01 deg; joints [35.963, -45.229, 108.255, -141.025, 69.06, 164.803]
  MoveL 8081 to (-134.08, 158.13, -64.5) mm, rotated rx -180 ry 0 rz 0.01 deg; joints [35.944, -45.232, 108.263, -141.046, 69.058, 164.813]
  MoveL 8082 to (-134.67, 157.06, -64.5) mm, rotated rx -180 ry 0 rz 0.01 deg; joints [35.896, -45.237, 108.276, -141.097, 69.051, 164.837]
  MoveL 8083 to (-134.95, 156.64, -64.5) mm, rotated rx -180 ry 0 rz 0.01 deg; joints [35.876, -45.237, 108.278, -141.118, 69.046, 164.845]
  MoveL 8084 to (-136.37, 154.8, -64.5) mm, rotated rx 180 ry 0 rz 0.01 deg; joints [35.784, -45.233, 108.271, -141.211, 69.018, 164.879]
  MoveL 8085 to (-136.62, 154.52, -64.5) mm, rotated rx -180 ry 0 rz 0.01 deg; joints [35.769, -45.231, 108.268, -141.226, 69.013, 164.883]
  MoveL 8086 to (-137.73, 153.36, -64.5) mm, rotated rx 180 ry 0 rz 0.01 deg; joints [35.707, -45.221, 108.247, -141.288, 68.987, 164.9]
  MoveL 8087 to (-138.02, 153.1, -64.5) mm, rotated rx 180 ry 0 rz 0.01 deg; joints [35.691, -45.217, 108.24, -141.303, 68.979, 164.903]
  MoveL 8088 to (-140.93, 150.73, -64.5) mm, rotated rx -180 ry 0 rz 0.01 deg; joints [35.549, -45.176, 108.151, -141.438, 68.902, 164.926]
  MoveL 8089 to (-141.16, 150.55, -64.5) mm, rotated rx 180 ry 0 rz 0.01 deg; joints [35.538, -45.172, 108.143, -141.449, 68.896, 164.927]
  MoveL 8090 to (-142.61, 149.57, -64.5) mm, rotated rx -180 ry 0 rz 0.01 deg; joints [35.473, -45.146, 108.089, -141.508, 68.855, 164.933]
  MoveL 8091 to (-142.82, 149.43, -64.5) mm, rotated rx 180 ry 0 rz 0.01 deg; joints [35.464, -45.142, 108.08, -141.517, 68.848, 164.933]
  MoveL 8092 to (-179.1, 128.45, -64.5) mm, rotated rx 180 ry 0 rz 0.01 deg; joints [33.977, -44.396, 106.459, -142.838, 67.736, 164.939]
  MoveC 8093 to (-179.56, 128.23, -64.5) mm, rotated rx 180 ry 0 rz 0.01 deg; joints [33.96, -44.386, 106.436, -142.852, 67.722, 164.938] to (-180.04, 128.08, -64.5) mm, rotated rx 180 ry 0 rz 0.01 deg; joints [33.944, -44.373, 106.407, -142.865, 67.705, 164.934]
  MoveL 8094 to (-181.13, 127.84, -64.5) mm, rotated rx 180 ry 0 rz 0.01 deg; joints [33.913, -44.341, 106.337, -142.888, 67.665, 164.922]
  MoveC 8095 to (-181.66, 127.76, -64.5) mm, rotated rx 180 ry 0 rz 0.01 deg; joints [33.898, -44.324, 106.301, -142.898, 67.645, 164.914] to (-182.2, 127.77, -64.5) mm, rotated rx -180 ry 0 rz 0.01 deg; joints [33.887, -44.306, 106.259, -142.904, 67.624, 164.904]
  MoveL 8096 to (-183.29, 127.87, -64.5) mm, rotated rx 180 ry 0 rz 0.01 deg; joints [33.867, -44.266, 106.171, -142.913, 67.58, 164.881]
  MoveC 8097 to (-183.83, 127.97, -64.5) mm, rotated rx 180 ry 0 rz 0.01 deg; joints [33.858, -44.246, 106.126, -142.915, 67.557, 164.868] to (-184.34, 128.15, -64.5) mm, rotated rx 180 ry 0 rz 0.01 deg; joints [33.853, -44.224, 106.078, -142.914, 67.534, 164.853]
  MoveL 8098 to (-185.37, 128.6, -64.5) mm, rotated rx -180 ry 0 rz 0.01 deg; joints [33.845, -44.179, 105.976, -142.908, 67.487, 164.819]
  MoveL 8099 to (-186.2, 129.12, -64.5) mm, rotated rx -180 ry 0 rz 0.01 deg; joints [33.844, -44.139, 105.887, -142.897, 67.448, 164.788]
  MoveL 8100 to (-186.85, 129.68, -64.5) mm, rotated rx -180 ry 0 rz 0.01 deg; joints [33.848, -44.105, 105.809, -142.882, 67.414, 164.758]
  MoveL 8101 to (-187.47, 130.37, -64.5) mm, rotated rx 180 ry 0 rz 0.01 deg; joints [33.857, -44.068, 105.727, -142.861, 67.38, 164.724]
  MoveL 8102 to (-188.05, 131.24, -64.5) mm, rotated rx 180 ry 0 rz 0.01 deg; joints [33.872, -44.029, 105.639, -142.833, 67.346, 164.686]
  MoveL 8103 to (-188.47, 132.11, -64.5) mm, rotated rx -180 ry 0 rz 0.01 deg; joints [33.891, -43.995, 105.563, -142.803, 67.317, 164.65]
  MoveL 8104 to (-188.75, 133, -64.5) mm, rotated rx 180 ry 0 rz 0.01 deg; joints [33.914, -43.966, 105.495, -142.769, 67.294, 164.616]
  MoveC 8105 to (-188.86, 133.5, -64.5) mm, rotated rx 180 ry 0 rz 0.01 deg; joints [33.928, -43.951, 105.461, -142.75, 67.282, 164.598] to (-188.9, 134.02, -64.5) mm, rotated rx -180 ry 0 rz 0.01 deg; joints [33.943, -43.938, 105.432, -142.73, 67.274, 164.58]
  MoveL 8106 to (-188.85, 267.36, -64.5) mm, rotated rx -180 ry 0 rz 0.01 deg; joints [38.012, -40.666, 98.024, -137.366, 65.433, 159.951]
  MoveL 8107 to (-204.67, 267.36, -64.5) mm, rotated rx 180 ry 0 rz 0.01 deg; joints [37.657, -40.099, 96.795, -137.522, 64.814, 159.614]
  MoveL 8108 to (-204.61, 134.02, -64.5) mm, rotated rx -180 ry 0 rz 0.01 deg; joints [33.607, -43.393, 104.226, -142.91, 66.65, 164.287]
  MoveC 8109 to (-204.65, 133.5, -64.5) mm, rotated rx 180 ry 0 rz 0.01 deg; joints [33.59, -43.403, 104.249, -142.931, 66.655, 164.303] to (-204.77, 133, -64.5) mm, rotated rx 180 ry 0 rz 0.01 deg; joints [33.571, -43.41, 104.266, -142.953, 66.657, 164.317]
  MoveL 8110 to (-205.05, 132.11, -64.5) mm, rotated rx -180 ry 0 rz 0.01 deg; joints [33.536, -43.42, 104.29, -142.993, 66.658, 164.341]
  MoveL 8111 to (-205.46, 131.24, -64.5) mm, rotated rx -180 ry 0 rz 0.01 deg; joints [33.5, -43.425, 104.302, -143.033, 66.653, 164.362]
  MoveL 8112 to (-206.04, 130.37, -64.5) mm, rotated rx -180 ry 0 rz 0.01 deg; joints [33.46, -43.424, 104.302, -143.075, 66.642, 164.379]
  MoveL 8113 to (-206.66, 129.68, -64.5) mm, rotated rx -180 ry 0 rz 0.01 deg; joints [33.425, -43.418, 104.289, -143.11, 66.627, 164.39]
  MoveL 8114 to (-207.32, 129.12, -64.5) mm, rotated rx -180 ry 0 rz 0.01 deg; joints [33.393, -43.407, 104.267, -143.14, 66.608, 164.395]
  MoveL 8115 to (-208.14, 128.6, -64.5) mm, rotated rx -180 ry 0 rz 0.01 deg; joints [33.359, -43.39, 104.23, -143.17, 66.582, 164.397]
  MoveL 8116 to (-209.17, 128.15, -64.5) mm, rotated rx -180 ry 0 rz 0.01 deg; joints [33.323, -43.363, 104.173, -143.2, 66.547, 164.392]
  MoveC 8117 to (-209.68, 127.97, -64.5) mm, rotated rx -180 ry 0 rz 0.01 deg; joints [33.306, -43.349, 104.142, -143.213, 66.529, 164.388] to (-210.22, 127.87, -64.5) mm, rotated rx -180 ry 0 rz 0.01 deg; joints [33.292, -43.333, 104.105, -143.223, 66.509, 164.381]
  MoveL 8118 to (-211.31, 127.77, -64.5) mm, rotated rx 180 ry 0 rz 0.01 deg; joints [33.265, -43.297, 104.026, -143.239, 66.466, 164.364]
  MoveC 8119 to (-211.85, 127.76, -64.5) mm, rotated rx 180 ry 0 rz 0.01 deg; joints [33.254, -43.278, 103.985, -143.245, 66.445, 164.354] to (-212.38, 127.84, -64.5) mm, rotated rx 180 ry 0 rz 0.01 deg; joints [33.245, -43.257, 103.939, -143.247, 66.422, 164.342]
  MoveL 8120 to (-213.47, 128.08, -64.5) mm, rotated rx -180 ry 0 rz 0.01 deg; joints [33.23, -43.213, 103.842, -143.249, 66.375, 164.313]
  MoveC 8121 to (-213.96, 128.23, -64.5) mm, rotated rx 180 ry 0 rz 0.01 deg; joints [33.225, -43.193, 103.796, -143.248, 66.353, 164.299] to (-214.41, 128.45, -64.5) mm, rotated rx 180 ry 0 rz 0.01 deg; joints [33.222, -43.172, 103.75, -143.244, 66.332, 164.284]
  MoveL 8122 to (-250.69, 149.43, -64.5) mm, rotated rx 180 ry 0 rz 0.01 deg; joints [33.136, -41.384, 99.79, -142.737, 64.571, 162.885]
  MoveL 8123 to (-250.95, 149.6, -64.5) mm, rotated rx 180 ry 0 rz 0.01 deg; joints [33.136, -41.371, 99.76, -142.733, 64.558, 162.874]
  MoveL 8124 to (-253.22, 151.2, -64.5) mm, rotated rx -180 ry 0 rz 0.01 deg; joints [33.139, -41.249, 99.492, -142.686, 64.442, 162.774]
  MoveL 8125 to (-253.46, 151.38, -64.5) mm, rotated rx -180 ry 0 rz 0.01 deg; joints [33.14, -41.237, 99.464, -142.681, 64.431, 162.763]
  MoveL 8126 to (-255.53, 153.13, -64.5) mm, rotated rx -180 ry 0 rz 0.01 deg; joints [33.153, -41.119, 99.203, -142.627, 64.321, 162.662]
  MoveL 8127 to (-255.84, 153.43, -64.5) mm, rotated rx -180 ry 0 rz 0.01 deg; joints [33.155, -41.1, 99.162, -142.617, 64.304, 162.645]
  MoveL 8128 to (-257.46, 155.19, -64.5) mm, rotated rx -180 ry 0 rz 0.01 deg; joints [33.177, -40.998, 98.937, -142.558, 64.213, 162.552]
  MoveL 8129 to (-257.75, 155.55, -64.5) mm, rotated rx -180 ry 0 rz 0.01 deg; joints [33.182, -40.979, 98.896, -142.546, 64.197, 162.534]
  MoveL 8130 to (-259.03, 157.39, -64.5) mm, rotated rx -180 ry 0 rz 0.01 deg; joints [33.213, -40.888, 98.694, -142.481, 64.119, 162.445]
  MoveL 8131 to (-259.33, 157.91, -64.5) mm, rotated rx 180 ry 0 rz 0.01 deg; joints [33.224, -40.865, 98.642, -142.462, 64.1, 162.42]
  MoveL 8132 to (-259.87, 159.09, -64.5) mm, rotated rx 180 ry 0 rz 0.01 deg; joints [33.249, -40.817, 98.535, -142.418, 64.062, 162.369]
  MoveL 8133 to (-260.03, 159.53, -64.5) mm, rotated rx -180 ry 0 rz 0.01 deg; joints [33.259, -40.8, 98.498, -142.401, 64.049, 162.35]
  MoveL 8134 to (-260.36, 160.61, -64.5) mm, rotated rx 180 ry 0 rz 0.01 deg; joints [33.286, -40.762, 98.413, -142.359, 64.021, 162.306]
  MoveL 8135 to (-260.49, 161.33, -64.5) mm, rotated rx 180 ry 0 rz 0.01 deg; joints [33.305, -40.74, 98.365, -142.33, 64.006, 162.278]
  MoveL 8136 to (-260.66, 163.5, -64.5) mm, rotated rx -180 ry 0 rz 0.01 deg; joints [33.369, -40.682, 98.234, -142.242, 63.969, 162.199]
  MoveL 8137 to (-260.65, 164.1, -64.5) mm, rotated rx 180 ry 0 rz 0.01 deg; joints [33.387, -40.668, 98.203, -142.217, 63.962, 162.179]
  MoveL 8138 to (-247.1, 299.4, -64.5) mm, rotated rx 180 ry 0 rz 0.01 deg; joints [37.638, -37.62, 91.398, -136.561, 62.671, 157.406]
  MoveL 8139 to (-247.09, 299.54, -64.5) mm, rotated rx -180 ry 0 rz 0.01 deg; joints [37.642, -37.617, 91.391, -136.556, 62.67, 157.401]
  MoveL 8140 to (-246.68, 302.44, -64.5) mm, rotated rx 180 ry 0 rz 0.01 deg; joints [37.731, -37.549, 91.24, -136.434, 62.647, 157.294]
  MoveL 8141 to (-246.63, 302.7, -64.5) mm, rotated rx -180 ry 0 rz 0.01 deg; joints [37.74, -37.543, 91.227, -136.423, 62.645, 157.284]
  MoveL 8142 to (-245.98, 305.6, -64.5) mm, rotated rx 180 ry 0 rz 0.01 deg; joints [37.834, -37.483, 91.095, -136.3, 62.631, 157.182]
  MoveL 8143 to (-245.92, 305.83, -64.5) mm, rotated rx 180 ry 0 rz 0.01 deg; joints [37.842, -37.479, 91.086, -136.29, 62.63, 157.174]
  MoveL 8144 to (-244.99, 309.01, -64.5) mm, rotated rx 180 ry 0 rz 0.01 deg; joints [37.951, -37.422, 90.959, -136.154, 62.625, 157.067]
  MoveL 8145 to (-244.91, 309.23, -64.5) mm, rotated rx 180 ry 0 rz 0.01 deg; joints [37.958, -37.419, 90.951, -136.144, 62.625, 157.06]
  MoveL 8146 to (-243.8, 312.22, -64.5) mm, rotated rx -180 ry 0 rz 0.01 deg; joints [38.065, -37.374, 90.85, -136.015, 62.629, 156.965]
  MoveL 8147 to (-243.56, 312.72, -64.5) mm, rotated rx -180 ry 0 rz 0.01 deg; joints [38.084, -37.368, 90.837, -135.992, 62.631, 156.95]
  MoveL 8148 to (-238.13, 322.16, -64.5) mm, rotated rx 180 ry 0 rz 0.01 deg; joints [38.463, -37.298, 90.673, -135.571, 62.721, 156.694]
  MoveL 8149 to (-237.79, 322.64, -64.5) mm, rotated rx 180 ry 0 rz 0.01 deg; joints [38.483, -37.296, 90.669, -135.549, 62.728, 156.682]
  MoveL 8150 to (-236.27, 324.45, -64.5) mm, rotated rx 180 ry 0 rz 0.01 deg; joints [38.566, -37.301, 90.675, -135.465, 62.764, 156.644]
  MoveL 8151 to (-235.98, 324.76, -64.5) mm, rotated rx 180 ry 0 rz 0.01 deg; joints [38.581, -37.303, 90.679, -135.45, 62.772, 156.639]
  MoveL 8152 to (-228.08, 332.09, -64.5) mm, rotated rx -180 ry 0 rz 0.01 deg; joints [38.956, -37.385, 90.845, -135.099, 62.988, 156.527]
  MoveL 8153 to (-227.65, 332.42, -64.5) mm, rotated rx -180 ry 0 rz 0.01 deg; joints [38.974, -37.391, 90.858, -135.082, 63, 156.523]
  MoveL 8154 to (-226.2, 333.39, -64.5) mm, rotated rx 180 ry 0 rz 0.01 deg; joints [39.033, -37.417, 90.912, -135.033, 63.045, 156.518]
  MoveL 8155 to (-225.79, 333.62, -64.5) mm, rotated rx -180 ry 0 rz 0.01 deg; joints [39.048, -37.426, 90.93, -135.02, 63.058, 156.518]
  MoveL 8156 to (-215.27, 338.66, -64.5) mm, rotated rx -180 ry 0 rz 0.01 deg; joints [39.42, -37.672, 91.45, -134.74, 63.408, 156.561]
  MoveL 8157 to (-214.72, 338.86, -64.5) mm, rotated rx 180 ry 0 rz 0.01 deg; joints [39.438, -37.686, 91.48, -134.728, 63.427, 156.566]
  MoveL 8158 to (-213.63, 339.17, -64.5) mm, rotated rx 180 ry 0 rz 0.01 deg; joints [39.471, -37.718, 91.548, -134.708, 63.466, 156.579]
  MoveL 8159 to (-213.49, 339.2, -64.5) mm, rotated rx -180 ry 0 rz 0.01 deg; joints [39.475, -37.722, 91.556, -134.705, 63.47, 156.581]
  MoveL 8160 to (-398.92, 339.2, -64.5) mm, rotated rx -180 ry 0 rz 0.01 deg; joints [35.657, -29.797, 74.752, -134.926, 55.444, 151.31]
  MoveL 8161 to (-400.13, 339.01, -64.5) mm, rotated rx -180 ry 0 rz 0.01 deg; joints [35.629, -29.744, 74.642, -134.927, 55.389, 151.277]
  MoveL 8162 to (-400.6, 338.83, -64.5) mm, rotated rx -180 ry 0 rz 0.01 deg; joints [35.615, -29.727, 74.607, -134.932, 55.37, 151.27]
  MoveL 8163 to (-401.11, 338.47, -64.33) mm, rotated rx -180 ry 0 rz 0.01 deg; joints [35.596, -29.722, 74.581, -134.943, 55.346, 151.264]
  MoveL 8164 to (-401.34, 338.07, -63.87) mm, rotated rx 180 ry 0 rz 0.01 deg; joints [35.581, -29.745, 74.59, -134.952, 55.329, 151.262]
  MoveL 8165 to (-401.39, 337.91, -63.23) mm, rotated rx 180 ry 0 rz 0.01 deg; joints [35.576, -29.776, 74.603, -134.949, 55.313, 151.248]
  Set speed (1000.0 mm/s)
  MoveL 8166 to (-401.39, 337.91, 11.77) mm, rotated rx 180 ry 0 rz 0.01 deg; joints [35.543, -32.957, 74.925, -133.511, 53.302, 148.747]
  Set speed (1000.0 mm/s)
  MoveL 8167 to (5.55, -23.88, 11.77) mm, rotated rx 180 ry 0 rz 0.01 deg; joints [32.85, -58.085, 126.976, -145.429, 72.999, 169.588]
  Set speed (100.0 mm/s)
  MoveL 8168 to (5.57, -23.72, 11.15) mm, rotated rx 180 ry 0 rz 0.01 deg; joints [32.857, -58.041, 126.97, -145.428, 73.031, 169.608]
  MoveL 8169 to (5.6, -23.27, 10.68) mm, rotated rx 180 ry 0 rz 0.01 deg; joints [32.876, -58.003, 126.952, -145.413, 73.051, 169.614]
  MoveL 8170 to (5.59, -22.66, 10.5) mm, rotated rx 180 ry 0 rz 0.01 deg; joints [32.899, -57.978, 126.924, -145.388, 73.054, 169.605]
  MoveL 8171 to (1.56, -17.42, 10.26) mm, rotated rx -180 ry 0 rz 0.01 deg; joints [33.002, -57.73, 126.425, -145.239, 72.869, 169.424]
  MoveL 8172 to (-4.85, -19.01, 10.01) mm, rotated rx 180 ry 0 rz 0.01 deg; joints [32.78, -57.539, 126.063, -145.437, 72.681, 169.391]
  MoveL 8173 to (-5.96, -25.52, 9.77) mm, rotated rx 180 ry 0 rz 0.01 deg; joints [32.499, -57.615, 126.269, -145.747, 72.731, 169.557]
  MoveL 8174 to (-0.44, -29.15, 9.52) mm, rotated rx -180 ry 0 rz 0.01 deg; joints [32.494, -57.847, 126.797, -145.803, 72.975, 169.733]
  MoveL 8175 to (5.09, -25.54, 9.28) mm, rotated rx 180 ry 0 rz 0.01 deg; joints [32.775, -57.939, 127.014, -145.538, 73.135, 169.72]
  MoveL 8176 to (4.01, -19.03, 9.04) mm, rotated rx -180 ry 0 rz 0.01 deg; joints [33.002, -57.761, 126.659, -145.275, 73.035, 169.545]
  MoveL 8177 to (-2.39, -17.41, 8.79) mm, rotated rx -180 ry 0 rz 0.01 deg; joints [32.904, -57.508, 126.157, -145.332, 72.811, 169.427]
  MoveL 8178 to (-6.44, -22.63, 8.55) mm, rotated rx -180 ry 0 rz 0.01 deg; joints [32.6, -57.464, 126.11, -145.642, 72.745, 169.521]
  MoveL 8179 to (-3.28, -28.43, 8.3) mm, rotated rx -180 ry 0 rz 0.01 deg; joints [32.453, -57.662, 126.573, -145.839, 72.934, 169.723]
  MoveL 8180 to (3.29, -27.86, 8.06) mm, rotated rx 180 ry 0 rz 0.01 deg; joints [32.64, -57.846, 126.992, -145.688, 73.166, 169.803]
  MoveL 8181 to (5.41, -21.6, 7.82) mm, rotated rx 180 ry 0 rz 0.01 deg; joints [32.938, -57.776, 126.863, -145.373, 73.178, 169.677]
  MoveL 8182 to (0.53, -17.16, 7.57) mm, rotated rx -180 ry 0 rz 0.01 deg; joints [32.988, -57.517, 126.341, -145.276, 72.972, 169.505]
  MoveL 8183 to (-5.5, -19.85, 7.33) mm, rotated rx -180 ry 0 rz 0.01 deg; joints [32.732, -57.361, 126.052, -145.515, 72.81, 169.506]
  MoveL 8184 to (-5.45, -26.45, 7.08) mm, rotated rx -180 ry 0 rz 0.01 deg; joints [32.477, -57.475, 126.34, -145.807, 72.901, 169.689]
  MoveL 8185 to (0.62, -29.05, 6.84) mm, rotated rx 180 ry 0 rz 0.01 deg; joints [32.526, -57.704, 126.862, -145.806, 73.153, 169.845]
  MoveL 8186 to (5.43, -24.53, 6.6) mm, rotated rx -180 ry 0 rz 0.01 deg; joints [32.825, -57.754, 126.99, -145.514, 73.278, 169.8]
  MoveL 8187 to (3.22, -18.31, 6.35) mm, rotated rx -180 ry 0 rz 0.01 deg; joints [33.012, -57.546, 126.571, -145.287, 73.142, 169.617]
  MoveL 8188 to (-3.37, -17.84, 6.11) mm, rotated rx -180 ry 0 rz 0.01 deg; joints [32.864, -57.311, 126.107, -145.398, 72.923, 169.527]
  MoveL 8189 to (-6.43, -23.69, 5.86) mm, rotated rx -180 ry 0 rz 0.01 deg; joints [32.561, -57.31, 126.153, -145.717, 72.9, 169.649]
  MoveL 8190 to (-2.3, -28.85, 5.62) mm, rotated rx 180 ry 0 rz 0.01 deg; joints [32.462, -57.526, 126.654, -145.866, 73.115, 169.847]
  MoveL 8191 to (4.07, -27.13, 5.37) mm, rotated rx 180 ry 0 rz 0.01 deg; joints [32.69, -57.68, 127.009, -145.668, 73.327, 169.896]
  MoveL 8192 to (5.05, -20.6, 5.13) mm, rotated rx 180 ry 0 rz 0.01 deg; joints [32.97, -57.569, 126.792, -145.363, 73.296, 169.748]
  MoveL 8193 to (-0.54, -17.08, 4.89) mm, rotated rx 180 ry 0 rz 0.01 deg; joints [32.966, -57.307, 126.262, -145.322, 73.075, 169.59]
  MoveL 8194 to (-6, -20.8, 4.64) mm, rotated rx 180 ry 0 rz 0.01 deg; joints [32.685, -57.189, 126.055, -145.594, 72.945, 169.624]
  MoveL 8195 to (-4.79, -27.29, 4.4) mm, rotated rx 180 ry 0 rz 0.01 deg; joints [32.463, -57.337, 126.417, -145.858, 73.076, 169.819]
  MoveL 8196 to (1.65, -28.78, 4.15) mm, rotated rx 180 ry 0 rz 0.01 deg; joints [32.565, -57.555, 126.915, -145.801, 73.328, 169.952]
  MoveL 8197 to (5.59, -23.48, 3.91) mm, rotated rx -180 ry 0 rz 0.01 deg; joints [32.872, -57.562, 126.951, -145.492, 73.413, 169.876]
  MoveL 8198 to (2.32, -17.74, 3.67) mm, rotated rx 180 ry 0 rz 0.01 deg; joints [33.013, -57.33, 126.481, -145.307, 73.245, 169.692]
  MoveL 8199 to (-4.25, -18.44, 3.42) mm, rotated rx 180 ry 0 rz 0.01 deg; joints [32.821, -57.12, 126.069, -145.469, 73.041, 169.632]
  MoveL 8200 to (-6.24, -24.74, 3.18) mm, rotated rx 180 ry 0 rz 0.01 deg; joints [32.527, -57.162, 126.207, -145.787, 73.06, 169.779]
  MoveL 8201 to (-1.27, -29.09, 2.93) mm, rotated rx 180 ry 0 rz 0.01 deg; joints [32.481, -57.388, 126.73, -145.884, 73.297, 169.967]
  MoveL 8202 to (4.71, -26.27, 2.69) mm, rotated rx -180 ry 0 rz 0.01 deg; joints [32.741, -57.507, 127.01, -145.645, 73.482, 169.983]
  MoveL 8203 to (4.53, -19.67, 2.45) mm, rotated rx -180 ry 0 rz 0.01 deg; joints [32.994, -57.358, 126.711, -145.361, 73.408, 169.818]
  MoveL 8204 to (-1.6, -17.2, 2.2) mm, rotated rx 180 ry 0 rz 0.01 deg; joints [32.937, -57.1, 126.191, -145.375, 73.181, 169.68]
  MoveL 8205 to (-6.32, -21.81, 1.96) mm, rotated rx -180 ry 0 rz 0.01 deg; joints [32.639, -57.023, 126.073, -145.672, 73.086, 169.747]
  MoveL 8206 to (-3.98, -27.99, 1.71) mm, rotated rx -180 ry 0 rz 0.01 deg; joints [32.457, -57.2, 126.497, -145.901, 73.254, 169.948]
  MoveL 8207 to (2.61, -28.32, 1.47) mm, rotated rx 180 ry 0 rz 0.01 deg; joints [32.609, -57.399, 126.955, -145.789, 73.499, 170.054]
  MoveL 8208 to (5.56, -22.41, 1.23) mm, rotated rx -180 ry 0 rz 0.01 deg; joints [32.915, -57.363, 126.898, -145.473, 73.542, 169.949]
  MoveL 8209 to (1.33, -17.34, 0.98) mm, rotated rx -180 ry 0 rz 0.01 deg; joints [33.005, -57.116, 126.392, -145.336, 73.347, 169.769]
  MoveL 8210 to (-5.01, -19.19, 0.74) mm, rotated rx 180 ry 0 rz 0.01 deg; joints [32.775, -56.935, 126.045, -145.544, 73.164, 169.741]
  MoveL 8211 to (-5.86, -25.74, 0.49) mm, rotated rx 180 ry 0 rz 0.01 deg; joints [32.499, -57.018, 126.271, -145.85, 73.226, 169.909]
  MoveL 8212 to (-0.2, -29.14, 0.25) mm, rotated rx 180 ry 0 rz 0.01 deg; joints [32.507, -57.246, 126.799, -145.892, 73.476, 170.083]
  MoveL 8213 to (5.19, -25.32, 0.01) mm, rotated rx -180 ry 0 rz 0.01 deg; joints [32.792, -57.326, 126.996, -145.62, 73.629, 170.065]
  MoveL 8214 to (3.84, -18.85, -0.24) mm, rotated rx 180 ry 0 rz 0.01 deg; joints [33.011, -57.144, 126.625, -145.365, 73.516, 169.888]
  MoveL 8215 to (-2.62, -17.49, -0.48) mm, rotated rx -180 ry 0 rz 0.01 deg; joints [32.901, -56.898, 126.13, -145.435, 73.29, 169.774]
  MoveL 8216 to (-6.46, -22.87, -0.73) mm, rotated rx -180 ry 0 rz 0.01 deg; joints [32.597, -56.864, 126.104, -145.748, 73.235, 169.872]
  MoveL 8217 to (-3.07, -28.54, -0.97) mm, rotated rx 180 ry 0 rz 0.01 deg; joints [32.46, -57.063, 126.577, -145.934, 73.434, 170.074]
  MoveL 8218 to (3.48, -27.71, -1.21) mm, rotated rx 180 ry 0 rz 0.01 deg; joints [32.657, -57.238, 126.982, -145.771, 73.664, 170.15]
  MoveL 8219 to (5.35, -21.37, -1.46) mm, rotated rx 180 ry 0 rz 0.01 deg; joints [32.952, -57.159, 126.832, -145.458, 73.663, 170.02]
  MoveL 8220 to (0.29, -17.12, -1.7) mm, rotated rx 180 ry 0 rz 0.01 deg; joints [32.989, -56.903, 126.307, -145.374, 73.449, 169.85]
  MoveL 8221 to (-5.63, -20.06, -1.95) mm, rotated rx -180 ry 0 rz 0.01 deg; joints [32.727, -56.757, 126.035, -145.621, 73.293, 169.855]
  MoveL 8222 to (-5.31, -26.66, -2.19) mm, rotated rx 180 ry 0 rz 0.01 deg; joints [32.479, -56.877, 126.341, -145.907, 73.398, 170.04]
  MoveL 8223 to (0.86, -29.01, -2.43) mm, rotated rx 180 ry 0 rz 0.01 deg; joints [32.541, -57.099, 126.859, -145.892, 73.654, 170.193]
  MoveL 8224 to (5.49, -24.3, -2.68) mm, rotated rx 180 ry 0 rz 0.01 deg; joints [32.842, -57.139, 126.966, -145.596, 73.769, 170.143]
  MoveL 8225 to (3.02, -18.17, -2.92) mm, rotated rx 180 ry 0 rz 0.01 deg; joints [33.019, -56.929, 126.534, -145.378, 73.62, 169.96]
  MoveL 8226 to (-3.58, -17.97, -3.17) mm, rotated rx 180 ry 0 rz 0.01 deg; joints [32.86, -56.702, 126.08, -145.502, 73.402, 169.873]
  MoveL 8227 to (-6.41, -23.94, -3.41) mm, rotated rx 180 ry 0 rz 0.01 deg; joints [32.558, -56.711, 126.147, -145.821, 73.39, 169.999]
  MoveL 8228 to (-2.07, -28.92, -3.65) mm, rotated rx -180 ry 0 rz 0.01 deg; joints [32.472, -56.925, 126.654, -145.958, 73.615, 170.196]
  MoveL 8229 to (4.23, -26.94, -3.9) mm, rotated rx 180 ry 0 rz 0.01 deg; joints [32.707, -57.069, 126.993, -145.749, 73.823, 170.24]
  MoveL 8230 to (4.95, -20.38, -4.14) mm, rotated rx 180 ry 0 rz 0.01 deg; joints [32.982, -56.951, 126.756, -145.449, 73.778, 170.089]
  MoveL 8231 to (-0.78, -17.09, -4.39) mm, rotated rx -180 ry 0 rz 0.01 deg; joints [32.965, -56.693, 126.228, -145.421, 73.552, 169.934]
  MoveL 8232 to (-6.09, -21.02, -4.63) mm, rotated rx 180 ry 0 rz 0.01 deg; joints [32.68, -56.585, 126.04, -145.699, 73.429, 169.973]
  MoveL 8233 to (-4.61, -27.46, -4.87) mm, rotated rx 180 ry 0 rz 0.01 deg; joints [32.466, -56.738, 126.417, -145.955, 73.573, 170.169]
  MoveL 8234 to (1.88, -28.69, -5.12) mm, rotated rx -180 ry 0 rz 0.01 deg; joints [32.58, -56.948, 126.907, -145.884, 73.827, 170.298]
  MoveL 8235 to (5.6, -23.24, -5.36) mm, rotated rx -180 ry 0 rz 0.01 deg; joints [32.888, -56.945, 126.921, -145.573, 73.901, 170.218]
  MoveL 8236 to (2.1, -17.64, -5.61) mm, rotated rx 180 ry 0 rz 0.01 deg; joints [33.018, -56.713, 126.442, -145.4, 73.722, 170.033]
  MoveL 8237 to (-4.43, -18.6, -5.85) mm, rotated rx 180 ry 0 rz 0.01 deg; joints [32.816, -56.511, 126.044, -145.573, 73.52, 169.977]
  MoveL 8238 to (-6.17, -24.98, -6.1) mm, rotated rx -180 ry 0 rz 0.01 deg; joints [32.525, -56.562, 126.202, -145.888, 73.552, 170.128]
  MoveL 8239 to (-1.02, -29.12, -6.34) mm, rotated rx -180 ry 0 rz 0.01 deg; joints [32.492, -56.785, 126.727, -145.972, 73.796, 170.314]
  MoveL 8240 to (4.83, -26.06, -6.58) mm, rotated rx 180 ry 0 rz 0.01 deg; joints [32.759, -56.893, 126.989, -145.724, 73.974, 170.326]
  MoveL 8241 to (4.38, -19.47, -6.83) mm, rotated rx -180 ry 0 rz 0.01 deg; joints [33.005, -56.738, 126.672, -145.447, 73.888, 170.158]
  MoveL 8242 to (-1.84, -17.25, -7.07) mm, rotated rx -180 ry 0 rz 0.01 deg; joints [32.935, -56.487, 126.157, -145.475, 73.657, 170.023]
  MoveL 8243 to (-6.37, -22.05, -7.32) mm, rotated rx 180 ry 0 rz 0.01 deg; joints [32.635, -56.42, 126.059, -145.776, 73.572, 170.094]
  MoveL 8244 to (-3.78, -28.13, -7.56) mm, rotated rx 180 ry 0 rz 0.01 deg; joints [32.463, -56.599, 126.495, -145.994, 73.752, 170.296]
  MoveL 8245 to (2.82, -28.2, -7.8) mm, rotated rx 180 ry 0 rz 0.01 deg; joints [32.625, -56.79, 126.942, -145.87, 73.996, 170.398]
  MoveL 8246 to (5.53, -22.17, -8.05) mm, rotated rx 180 ry 0 rz 0.01 deg; joints [32.929, -56.744, 126.863, -145.554, 74.026, 170.289]
  MoveL 8247 to (1.1, -17.28, -8.29) mm, rotated rx 180 ry 0 rz 0.01 deg; joints [33.008, -56.498, 126.352, -145.43, 73.823, 170.11]
  MoveL 8248 to (-5.17, -19.38, -8.54) mm, rotated rx 180 ry 0 rz 0.01 deg; joints [32.77, -56.327, 126.021, -145.647, 73.644, 170.086]
  MoveL 8249 to (-5.75, -25.96, -8.78) mm, rotated rx 180 ry 0 rz 0.01 deg; joints [32.499, -56.417, 126.265, -145.949, 73.719, 170.257]
  MoveL 8250 to (0.04, -29.13, -9.02) mm, rotated rx -180 ry 0 rz 0.01 deg; joints [32.52, -56.64, 126.792, -145.977, 73.975, 170.428]
  MoveL 8251 to (5.27, -25.09, -9.27) mm, rotated rx 180 ry 0 rz 0.01 deg; joints [32.809, -56.71, 126.969, -145.699, 74.119, 170.406]
  MoveL 8252 to (3.67, -18.68, -9.51) mm, rotated rx 180 ry 0 rz 0.01 deg; joints [33.019, -56.524, 126.582, -145.452, 73.994, 170.228]
  MoveL 8253 to (-2.85, -17.59, -9.76) mm, rotated rx -180 ry 0 rz 0.01 deg; joints [32.898, -56.286, 126.096, -145.535, 73.766, 170.117]
  MoveL 8254 to (-6.46, -23.11, -10) mm, rotated rx -180 ry 0 rz 0.01 deg; joints [32.593, -56.261, 126.091, -145.85, 73.722, 170.218]
  MoveC 8255 to (-4.82, -27.08, -10) mm, rotated rx 180 ry 0 rz 0.01 deg; joints [32.48, -56.387, 126.373, -145.992, 73.83, 170.344] to (-0.85, -28.72, -10) mm, rotated rx -180 ry 0 rz 0.01 deg; joints [32.514, -56.54, 126.711, -145.986, 73.99, 170.441]
  MoveC 8256 to (3.11, -27.08, -10) mm, rotated rx 180 ry 0 rz 0.01 deg; joints [32.678, -56.632, 126.907, -145.836, 74.107, 170.454] to (4.75, -23.11, -10) mm, rotated rx -180 ry 0 rz 0.01 deg; joints [32.874, -56.609, 126.846, -145.629, 74.114, 170.375]
  MoveL 8257 to (4.75, -20.36, -10) mm, rotated rx 180 ry 0 rz 0.01 deg; joints [32.982, -56.557, 126.727, -145.509, 74.078, 170.304]
  MoveC 8258 to (3.65, -18.8, -10) mm, rotated rx -180 ry 0 rz 0.01 deg; joints [33.015, -56.493, 126.585, -145.462, 74.02, 170.248] to (1.8, -19.32, -10) mm, rotated rx -180 ry 0 rz 0.01 deg; joints [32.948, -56.446, 126.484, -145.522, 73.962, 170.236]
  MoveL 8259 to (-0.81, -22.56, -10) mm, rotated rx 180 ry 0 rz 0.01 deg; joints [32.756, -56.426, 126.448, -145.715, 73.913, 170.283]
  MoveC 8260 to (-1.05, -24.63, -10) mm, rotated rx -180 ry 0 rz 0.01 deg; joints [32.669, -56.458, 126.522, -145.811, 73.931, 170.333] to (0.71, -25.74, -10) mm, rotated rx -180 ry 0 rz 0.01 deg; joints [32.67, -56.533, 126.688, -145.825, 74.006, 170.386]
  MoveL 8261 to (2.64, -25.74, -10) mm, rotated rx 180 ry 0 rz 0.01 deg; joints [32.718, -56.593, 126.818, -145.787, 74.074, 170.413]
  MoveC 8262 to (4.13, -25.12, -10) mm, rotated rx -180 ry 0 rz 0.01 deg; joints [32.78, -56.627, 126.892, -145.73, 74.118, 170.418] to (4.75, -23.63, -10) mm, rotated rx 180 ry 0 rz 0.01 deg; joints [32.854, -56.618, 126.869, -145.652, 74.12, 170.389]
  MoveL 8263 to (4.75, -23.11, -10) mm, rotated rx -180 ry 0 rz 0.01 deg; joints [32.874, -56.609, 126.846, -145.629, 74.114, 170.375]
  MoveL 8264 to (3.54, -23.38, -10) mm, rotated rx 180 ry 0 rz 0.01 deg; joints [32.833, -56.576, 126.776, -145.665, 74.075, 170.365]
  MoveL 8265 to (4.03, -24.45, -10) mm, rotated rx 180 ry 0 rz 0.01 deg; joints [32.804, -56.611, 126.856, -145.702, 74.106, 170.399]
  MoveL 8266 to (4.23, -24.69, -10) mm, rotated rx 180 ry 0 rz 0.01 deg; joints [32.799, -56.622, 126.879, -145.709, 74.116, 170.408]
  MoveL 8267 to (8.68, -28.03, -10) mm, rotated rx -180 ry 0 rz 0.01 deg; joints [32.781, -56.821, 127.322, -145.766, 74.313, 170.556]
  MoveL 8268 to (9.37, -28.67, -10) mm, rotated rx 180 ry 0 rz 0.01 deg; joints [32.773, -56.854, 127.396, -145.781, 74.346, 170.582]
  MoveL 8269 to (9.68, -28.6, -10) mm, rotated rx 180 ry 0 rz 0.01 deg; joints [32.784, -56.863, 127.414, -145.772, 74.355, 170.585]
  MoveL 8270 to (10.02, -27.8, -10) mm, rotated rx 180 ry 0 rz 0.01 deg; joints [32.824, -56.858, 127.402, -145.729, 74.357, 170.569]
  MoveL 8271 to (10.22, -26.94, -10) mm, rotated rx -180 ry 0 rz 0.01 deg; joints [32.863, -56.848, 127.378, -145.688, 74.353, 170.55]
  MoveL 8272 to (10.27, -25.87, -10) mm, rotated rx -180 ry 0 rz 0.01 deg; joints [32.906, -56.83, 127.336, -145.639, 74.341, 170.523]
  MoveL 8273 to (10.27, 7.53, -10) mm, rotated rx -180 ry 0 rz 0.01 deg; joints [34.198, -56.188, 125.86, -144.186, 73.911, 169.65]
  MoveL 8274 to (6.2, -2.88, -10) mm, rotated rx 180 ry 0 rz 0.01 deg; joints [33.695, -56.267, 126.055, -144.719, 73.904, 169.868]
  MoveL 8275 to (5.98, -3.35, -10) mm, rotated rx -180 ry 0 rz 0.01 deg; joints [33.671, -56.269, 126.061, -144.743, 73.903, 169.877]
  MoveL 8276 to (1.99, -10.24, -10) mm, rotated rx -180 ry 0 rz 0.01 deg; joints [33.304, -56.279, 126.098, -145.122, 73.853, 170.002]
  MoveL 8277 to (1.69, -10.67, -10) mm, rotated rx -180 ry 0 rz 0.01 deg; joints [33.28, -56.278, 126.097, -145.147, 73.848, 170.009]
  MoveL 8278 to (-6.46, -20.77, -10) mm, rotated rx 180 ry 0 rz 0.01 deg; joints [32.684, -56.217, 125.989, -145.747, 73.692, 170.158]
  MoveL 8279 to (-7.17, -21.43, -10) mm, rotated rx -180 ry 0 rz 0.01 deg; joints [32.641, -56.208, 125.97, -145.79, 73.676, 170.165]
  MoveL 8280 to (-10.54, -23.75, -10) mm, rotated rx -180 ry 0 rz 0.01 deg; joints [32.467, -56.146, 125.842, -145.957, 73.587, 170.178]
  MoveL 8281 to (-10.6, -23.8, -10) mm, rotated rx 180 ry 0 rz 0.01 deg; joints [32.464, -56.145, 125.84, -145.96, 73.585, 170.178]
  MoveL 8282 to (-18.17, -28.78, -10) mm, rotated rx 180 ry 0 rz 0.01 deg; joints [32.084, -56.001, 125.539, -146.322, 73.381, 170.202]
  MoveL 8283 to (-18.86, -29.13, -10) mm, rotated rx -180 ry 0 rz 0.01 deg; joints [32.054, -55.986, 125.507, -146.351, 73.361, 170.201]
  MoveL 8284 to (-20, -29.55, -10) mm, rotated rx -180 ry 0 rz 0.01 deg; joints [32.01, -55.958, 125.447, -146.39, 73.326, 170.196]
  MoveL 8285 to (-20.24, -29.63, -10) mm, rotated rx -180 ry 0 rz 0.01 deg; joints [32.001, -55.952, 125.434, -146.398, 73.319, 170.195]
  MoveL 8286 to (-26, -31.27, -10) mm, rotated rx -180 ry 0 rz 0.01 deg; joints [31.798, -55.801, 125.109, -146.578, 73.135, 170.157]
  MoveL 8287 to (5.41, -31.27, -10) mm, rotated rx 180 ry 0 rz 0.01 deg; joints [32.571, -56.781, 127.242, -145.974, 74.241, 170.593]
  MoveL 8288 to (6.62, -31.07, -10) mm, rotated rx -180 ry 0 rz 0.01 deg; joints [32.609, -56.815, 127.315, -145.942, 74.281, 170.605]
  Set speed (1000.0 mm/s)
  MoveL 8289 to (6.62, -31.07, 11) mm, rotated rx 180 ry 0 rz 0.01 deg; joints [32.595, -58.209, 127.357, -145.734, 73.159, 169.819]
  Set speed (1000.0 mm/s)
  MoveL 8290 to (5.57, -23.89, 11) mm, rotated rx -180 ry 0 rz 0.01 deg; joints [32.85, -58.035, 126.977, -145.438, 73.04, 169.618]
  Set speed (1000.0 mm/s)
  MoveL 8291 to (5.57, -23.89, 1.77) mm, rotated rx 180 ry 0 rz 0.01 deg; joints [32.856, -57.427, 126.963, -145.532, 73.531, 169.967]
  Set speed (100.0 mm/s)
  MoveL 8292 to (5.58, -23.73, 1.15) mm, rotated rx 180 ry 0 rz 0.01 deg; joints [32.864, -57.384, 126.956, -145.531, 73.563, 169.987]
  MoveL 8293 to (5.61, -23.29, 0.68) mm, rotated rx -180 ry 0 rz 0.01 deg; joints [32.882, -57.346, 126.938, -145.516, 73.583, 169.993]
  MoveL 8294 to (5.6, -22.67, 0.5) mm, rotated rx 180 ry 0 rz 0.01 deg; joints [32.906, -57.321, 126.91, -145.491, 73.584, 169.984]
  MoveL 8295 to (1.57, -17.43, 0.26) mm, rotated rx -180 ry 0 rz 0.01 deg; joints [33.008, -57.077, 126.411, -145.343, 73.395, 169.802]
  MoveL 8296 to (-4.84, -19.02, 0.01) mm, rotated rx 180 ry 0 rz 0.01 deg; joints [32.786, -56.89, 126.048, -145.541, 73.206, 169.766]
  MoveL 8297 to (-5.95, -25.53, -0.23) mm, rotated rx 180 ry 0 rz 0.01 deg; joints [32.505, -56.963, 126.254, -145.85, 73.259, 169.93]
  MoveL 8298 to (-0.43, -29.16, -0.48) mm, rotated rx -180 ry 0 rz 0.01 deg; joints [32.501, -57.191, 126.782, -145.905, 73.507, 170.107]
  MoveL 8299 to (5.1, -25.56, -0.72) mm, rotated rx -180 ry 0 rz 0.01 deg; joints [32.781, -57.28, 126.999, -145.64, 73.667, 170.098]
  MoveL 8300 to (4.02, -19.04, -0.96) mm, rotated rx 180 ry 0 rz 0.01 deg; joints [33.008, -57.105, 126.643, -145.377, 73.563, 169.923]
  MoveL 8301 to (-2.38, -17.42, -1.21) mm, rotated rx 180 ry 0 rz 0.01 deg; joints [32.91, -56.857, 126.142, -145.435, 73.335, 169.803]
  MoveL 8302 to (-6.43, -22.64, -1.45) mm, rotated rx 180 ry 0 rz 0.01 deg; joints [32.607, -56.813, 126.094, -145.745, 73.271, 169.893]
  MoveL 8303 to (-3.27, -28.44, -1.7) mm, rotated rx -180 ry 0 rz 0.01 deg; joints [32.459, -57.007, 126.557, -145.941, 73.464, 170.095]
  MoveL 8304 to (3.31, -27.87, -1.94) mm, rotated rx -180 ry 0 rz 0.01 deg; joints [32.646, -57.187, 126.976, -145.789, 73.698, 170.179]
  MoveL 8305 to (5.42, -21.62, -2.18) mm, rotated rx -180 ry 0 rz 0.01 deg; joints [32.944, -57.118, 126.847, -145.475, 73.707, 170.055]
  MoveL 8306 to (0.54, -17.17, -2.43) mm, rotated rx 180 ry 0 rz 0.01 deg; joints [32.994, -56.864, 126.325, -145.379, 73.496, 169.881]
  MoveL 8307 to (-5.49, -19.86, -2.67) mm, rotated rx -180 ry 0 rz 0.01 deg; joints [32.739, -56.71, 126.035, -145.617, 73.333, 169.878]
  MoveL 8308 to (-5.44, -26.47, -2.92) mm, rotated rx 180 ry 0 rz 0.01 deg; joints [32.483, -56.821, 126.323, -145.908, 73.429, 170.06]
  MoveL 8309 to (0.63, -29.07, -3.16) mm, rotated rx -180 ry 0 rz 0.01 deg; joints [32.533, -57.045, 126.844, -145.907, 73.685, 170.218]
  MoveL 8310 to (5.44, -24.55, -3.4) mm, rotated rx 180 ry 0 rz 0.01 deg; joints [32.831, -57.094, 126.972, -145.615, 73.809, 170.177]
  MoveL 8311 to (3.23, -18.33, -3.65) mm, rotated rx 180 ry 0 rz 0.01 deg; joints [33.018, -56.89, 126.553, -145.388, 73.668, 169.994]
  MoveL 8312 to (-3.36, -17.86, -3.89) mm, rotated rx -180 ry 0 rz 0.01 deg; joints [32.871, -56.659, 126.089, -145.5, 73.447, 169.9]
  MoveL 8313 to (-6.42, -23.71, -4.14) mm, rotated rx 180 ry 0 rz 0.01 deg; joints [32.567, -56.658, 126.135, -145.818, 73.425, 170.02]
  MoveL 8314 to (-2.29, -28.86, -4.38) mm, rotated rx 180 ry 0 rz 0.01 deg; joints [32.469, -56.869, 126.635, -145.967, 73.645, 170.218]
  MoveL 8315 to (4.08, -27.14, -4.63) mm, rotated rx 180 ry 0 rz 0.01 deg; joints [32.696, -57.02, 126.99, -145.768, 73.858, 170.27]
  MoveL 8316 to (5.06, -20.61, -4.87) mm, rotated rx 180 ry 0 rz 0.01 deg; joints [32.976, -56.911, 126.773, -145.464, 73.823, 170.124]
  MoveL 8317 to (-0.53, -17.1, -5.11) mm, rotated rx -180 ry 0 rz 0.01 deg; joints [32.972, -56.653, 126.243, -145.423, 73.599, 169.965]
  MoveL 8318 to (-5.99, -20.81, -5.36) mm, rotated rx 180 ry 0 rz 0.01 deg; joints [32.691, -56.537, 126.036, -145.695, 73.468, 169.995]
  MoveL 8319 to (-4.77, -27.3, -5.6) mm, rotated rx -180 ry 0 rz 0.01 deg; joints [32.469, -56.682, 126.397, -145.958, 73.604, 170.189]
  MoveL 8320 to (1.66, -28.79, -5.85) mm, rotated rx -180 ry 0 rz 0.01 deg; joints [32.571, -56.895, 126.895, -145.9, 73.859, 170.325]
  MoveL 8321 to (5.6, -23.49, -6.09) mm, rotated rx 180 ry 0 rz 0.01 deg; joints [32.878, -56.901, 126.931, -145.591, 73.942, 170.252]
  MoveL 8322 to (2.33, -17.76, -6.33) mm, rotated rx -180 ry 0 rz 0.01 deg; joints [33.019, -56.675, 126.461, -145.408, 73.77, 170.067]
  MoveL 8323 to (-4.24, -18.46, -6.58) mm, rotated rx -180 ry 0 rz 0.01 deg; joints [32.827, -56.467, 126.049, -145.57, 73.563, 170.003]
  MoveL 8324 to (-6.23, -24.76, -6.82) mm, rotated rx -180 ry 0 rz 0.01 deg; joints [32.533, -56.508, 126.186, -145.887, 73.585, 170.148]
  MoveL 8325 to (-1.25, -29.1, -7.07) mm, rotated rx 180 ry 0 rz 0.01 deg; joints [32.487, -56.729, 126.709, -145.983, 73.826, 170.338]
  MoveL 8326 to (4.72, -26.29, -7.31) mm, rotated rx 180 ry 0 rz 0.01 deg; joints [32.747, -56.846, 126.989, -145.743, 74.011, 170.357]
  MoveL 8327 to (4.54, -19.69, -7.55) mm, rotated rx -180 ry 0 rz 0.01 deg; joints [33.001, -56.699, 126.69, -145.46, 73.934, 170.193]
  MoveL 8328 to (-1.59, -17.21, -7.8) mm, rotated rx 180 ry 0 rz 0.01 deg; joints [32.943, -56.446, 126.17, -145.475, 73.703, 170.052]
  MoveL 8329 to (-6.31, -21.83, -8.04) mm, rotated rx 180 ry 0 rz 0.01 deg; joints [32.646, -56.37, 126.051, -145.772, 73.609, 170.116]
  MoveL 8330 to (-3.97, -28, -8.29) mm, rotated rx 180 ry 0 rz 0.01 deg; joints [32.463, -56.543, 126.475, -145.999, 73.781, 170.317]
  MoveL 8331 to (2.62, -28.34, -8.53) mm, rotated rx 180 ry 0 rz 0.01 deg; joints [32.615, -56.738, 126.933, -145.887, 74.029, 170.425]
  MoveL 8332 to (5.57, -22.43, -8.77) mm, rotated rx 180 ry 0 rz 0.01 deg; joints [32.921, -56.702, 126.875, -145.571, 74.069, 170.324]
  MoveL 8333 to (1.34, -17.36, -9.02) mm, rotated rx 180 ry 0 rz 0.01 deg; joints [33.012, -56.459, 126.37, -145.436, 73.87, 170.142]
  MoveL 8334 to (-5, -19.2, -9.26) mm, rotated rx -180 ry 0 rz 0.01 deg; joints [32.781, -56.282, 126.022, -145.643, 73.685, 170.111]
  MoveL 8335 to (-5.85, -25.75, -9.51) mm, rotated rx -180 ry 0 rz 0.01 deg; joints [32.505, -56.362, 126.247, -145.949, 73.751, 170.277]
  MoveL 8336 to (-0.19, -29.16, -9.75) mm, rotated rx 180 ry 0 rz 0.01 deg; joints [32.513, -56.585, 126.775, -145.99, 74.005, 170.452]
  MoveL 8337 to (5.2, -25.33, -9.99) mm, rotated rx 180 ry 0 rz 0.01 deg; joints [32.799, -56.664, 126.972, -145.718, 74.157, 170.438]
  MoveL 8338 to (3.85, -18.87, -10.24) mm, rotated rx 180 ry 0 rz 0.01 deg; joints [33.017, -56.485, 126.601, -145.464, 74.04, 170.262]
  MoveL 8339 to (-2.61, -17.51, -10.48) mm, rotated rx 180 ry 0 rz 0.01 deg; joints [32.907, -56.244, 126.106, -145.534, 73.81, 170.145]
  MoveL 8340 to (-6.45, -22.88, -10.73) mm, rotated rx 180 ry 0 rz 0.01 deg; joints [32.603, -56.21, 126.08, -145.847, 73.757, 170.239]
  MoveL 8341 to (-3.06, -28.55, -10.97) mm, rotated rx 180 ry 0 rz 0.01 deg; joints [32.466, -56.405, 126.552, -146.031, 73.961, 170.441]
  MoveL 8342 to (3.49, -27.72, -11.21) mm, rotated rx -180 ry 0 rz 0.01 deg; joints [32.663, -56.575, 126.957, -145.868, 74.193, 170.521]
  MoveL 8343 to (5.36, -21.38, -11.46) mm, rotated rx 180 ry 0 rz 0.01 deg; joints [32.958, -56.498, 126.807, -145.555, 74.189, 170.393]
  MoveL 8344 to (0.3, -17.14, -11.7) mm, rotated rx 180 ry 0 rz 0.01 deg; joints [32.996, -56.246, 126.282, -145.473, 73.97, 170.221]
  MoveL 8345 to (-5.62, -20.07, -11.95) mm, rotated rx -180 ry 0 rz 0.01 deg; joints [32.734, -56.103, 126.01, -145.719, 73.814, 170.223]
  MoveL 8346 to (-5.3, -26.67, -12.19) mm, rotated rx -180 ry 0 rz 0.01 deg; joints [32.485, -56.22, 126.316, -146.004, 73.922, 170.406]
  MoveL 8347 to (0.87, -29.02, -12.43) mm, rotated rx -180 ry 0 rz 0.01 deg; joints [32.547, -56.437, 126.833, -145.988, 74.182, 170.562]
  MoveL 8348 to (5.5, -24.31, -12.68) mm, rotated rx -180 ry 0 rz 0.01 deg; joints [32.848, -56.476, 126.94, -145.692, 74.296, 170.515]
  MoveL 8349 to (3.03, -18.18, -12.92) mm, rotated rx 180 ry 0 rz 0.01 deg; joints [33.025, -56.269, 126.508, -145.475, 74.143, 170.332]
  MoveL 8350 to (-3.57, -17.98, -13.17) mm, rotated rx -180 ry 0 rz 0.01 deg; joints [32.867, -56.047, 126.054, -145.6, 73.922, 170.242]
  MoveL 8351 to (-6.39, -23.95, -13.41) mm, rotated rx 180 ry 0 rz 0.01 deg; joints [32.565, -56.055, 126.121, -145.918, 73.912, 170.365]
  MoveL 8352 to (-2.06, -28.93, -13.65) mm, rotated rx 180 ry 0 rz 0.01 deg; joints [32.478, -56.265, 126.627, -146.053, 74.142, 170.563]
  MoveL 8353 to (4.24, -26.96, -13.9) mm, rotated rx -180 ry 0 rz 0.01 deg; joints [32.714, -56.405, 126.966, -145.845, 74.35, 170.61]
  MoveL 8354 to (4.96, -20.39, -14.14) mm, rotated rx -180 ry 0 rz 0.01 deg; joints [32.988, -56.289, 126.729, -145.545, 74.302, 170.461]
  MoveL 8355 to (-0.77, -17.11, -14.39) mm, rotated rx -180 ry 0 rz 0.01 deg; joints [32.972, -56.036, 126.2, -145.518, 74.072, 170.304]
  MoveL 8356 to (-6.08, -21.04, -14.63) mm, rotated rx -180 ry 0 rz 0.01 deg; joints [32.687, -55.93, 126.012, -145.796, 73.949, 170.339]
  MoveL 8357 to (-4.6, -27.47, -14.87) mm, rotated rx 180 ry 0 rz 0.01 deg; joints [32.473, -56.079, 126.389, -146.051, 74.097, 170.534]
  MoveL 8358 to (1.89, -28.7, -15.12) mm, rotated rx 180 ry 0 rz 0.01 deg; joints [32.587, -56.284, 126.879, -145.979, 74.354, 170.666]
